Omron Sysmac Studio project Bowery_Farm1 (Sysmac Studio 1.47.0.64008, StandardProject)

# Controller Bowery_Farm1: NJ101-9000 version 1.14
Units and slaves: Node1 : NX-ECC203 (E001); Unit 1 : NX-OD5121 (N1); Unit 2 : NX-SID800 (N2); Unit 3 : NX-SOD400 (N3); Node41 : GX-JC06(IN,X2,X3) Main device (E005); Node8 : NX-ECC203 (LiftGR04); Unit 1 : NX-ID5442 (N9_1); Unit 2 : NX-ID5442 (N10_1); Unit 3 : NX-OD4121 (N11_1); Unit 4 : NX-SID800 (N12_1); Unit 5 : NX-SOD400 (N13_1); Node42 : GX-JC03 (E003); Node43 : NX-ECC203 (E004); Unit 1 : NX-EC0222 (N8_1); Node5 : NX-ECC203 (LiftGR03); Unit 1 : NX-ID5442 (N9); Unit 2 : NX-ID5442 (N10); Unit 3 : NX-OD4121 (N11); Unit 4 : NX-SID800 (N12); Unit 5 : NX-SOD400 (N13); Node32 : GX-JC03 (LiftGR03_Switch); Node33 : NX-ECC203 (LiftGR03_Dek); Unit 1 : NX-EC0222 (N33); Node44 : GX-JC06(X4,X5,X6) Sub-device (E006); Power Supply : NJ-Px3001; CPU : NJ101-9000
Task PrimaryTask (priority 4, period or condition 4000): Mobile_Machines, General, Work_Level01, Work_Mezzanine
Task ReadSettings (priority 8, period or condition 20000): ReadSettings
Library Greencube library 1.2020.1116 (contents left out)

TYPE ST_FB_40401_InputsLift : STRUCT
    LS_FallProtect : BOOL;  (* Limit switch fall protection *)
    LS_Lift_Up : BOOL;  (* Limit switch lift up *)
    LS_Lift_Down : BOOL;  (* Limit switch lift down *)
    LC_Car_Free_Back : BOOL;  (* Photocell carrier detection free backside *)
    LC_Car_Present : BOOL;  (* Photocell carrier present *)
    LC_Car_Free_Front : BOOL;  (* Photocell carrier detection free frontside *)
    LC_Con_Free_Back : BOOL;  (* Photocell container detection free backside *)
    LC_Con_Present : BOOL;  (* Photocell container present *)
    LC_Con_Free_Front : BOOL;  (* Photocell container detection free frontside *)
    IS_Act_Back_Out : BOOL;  (* Inductive sensor actuator backside out *)
    IS_Act_Back_In : BOOL;  (* Inductive sensor actuator backside in *)
    IS_Act_Front_Out : BOOL;  (* Inductive sensor actuator frontside out *)
    IS_Act_Front_In : BOOL;  (* Inductive sensor actuator frontside in *)
    IS_Lift_Level : BOOL;  (* Inductive sensor lift at a level *)
    Clixon_M1 : BOOL;  (* Temperature controller M1 *)
    Clixon_M2 : BOOL;  (* Temperature controller M2 *)
    Clixon_M3 : BOOL;  (* Temperature controller M3 *)
    Clixon_M4 : BOOL;  (* Temperature controller M4 *)
    RC_Tray_Stopper_Min_Back_Up : BOOL;  (* Tray stopper min backside *)
    RC_Tray_Stopper_Max_Back_Up : BOOL;  (* Tray stopper max backside *)
    RC_Tray_Stopper_Min_Front_Up : BOOL;  (* Tray stopper min frontside *)
    RC_Tray_Stopper_Max_Front_Up : BOOL;  (* Tray stopper max frontside *)
    IS_Con_In_Pos_Front : BOOL;  (* Inductive sensor tray is in position front *)
    IS_Con_In_Pos_Back : BOOL;  (* Inductive sensor tray is in position back *)
    LC_Lift_Free_Back : ARRAY[0..15] OF BOOL;  (* Photocell lift free backside Level[i] *)
    LC_Lift_Free_Front : ARRAY[0..15] OF BOOL;  (* Photocell lift free frontside Level[i] *)
    IO_OK : BOOL;  (* Ethercat IO is OK *)
END_STRUCT END_TYPE
TYPE ST_FB_40303_Commands : STRUCT
    SprayBoomToLeft : BOOL;  (* Move sprayboom to left; offset 0.0 *)
    SprayBoomToRight : BOOL;  (* Move sprayboom to right; offset 0.1 *)
    SprayBoomStop : BOOL;  (* Move sprayboom stop; offset 0.2 *)
    LiftingFrame_Up : BOOL;  (* Lifting frame up; offset 1.0 *)
    LiftingFrame_Down : BOOL;  (* Lifting frame down; offset 1.1 *)
    LiftingFrameFirstPush_Up : BOOL;  (* Lifting frame first push up; offset 2.0 *)
    LiftingFrameFirstPush_Down : BOOL;  (* Lifting frame first push down; offset 2.1 *)
    ClampsContainerClose : BOOL;  (* Clamps container close; offset 3.0 *)
    ClampsContainerOpen : BOOL;  (* Clamps container open; offset 3.1 *)
    ClampsBottomLeft_Up : BOOL;  (* Clamps bottom left up; offset 4.0 *)
    ClampsBottomLeft_Down : BOOL;  (* Clamps bottom left down; offset 4.1 *)
    ClampsBottomRight_Up : BOOL;  (* Clamps bottom right up; offset 5.0 *)
    ClampsBottomRight_Down : BOOL;  (* Clamps bottom right down; offset 5.1 *)
    DirtBelt_Forward : BOOL;  (* Dirtbelt forward; offset 6.0 *)
    DirtBelt_Backward : BOOL;  (* Dirtbelt backward; offset 6.1 *)
    DirtBelt_Stop : BOOL;  (* Dirtbelt stop; offset 6.2 *)
    Brush_Forward : BOOL;  (* Brush forward; offset 7.0 *)
    Brush_Backward : BOOL;  (* Brush backward; offset 7.1 *)
    Brush_Stop : BOOL;  (* Brush stop; offset 7.2 *)
    Brush_Fixed : BOOL;  (* Brush fixed; offset 8.0 *)
    Brush_Loose : BOOL;  (* Brush loose; offset 8.1 *)
    SemiAutomatic_StartWashCycle : BOOL;  (* SemiAutomatic, start wash cycle; offset 9.0 *)
    SemiAutomatic_StartCleanBrushCycle : BOOL;  (* SemiAutomatic, start clean brush cycle; offset 9.1 *)
END_STRUCT END_TYPE
TYPE ST_FB_40303_Inputs : STRUCT
    EmergencyStop_OK : BOOL;  (* Emergency stop OK *)
    TurningFrame_Up : BOOL;  (* Lifting frame cilinder is out *)
    TurningFrame_Middle : BOOL;  (* Lifting frame cilinder is in *)
    TurningFrame_Down : BOOL;  (* Lifting frame cilinder is out *)
    Container_Present_1 : BOOL;  (* Container present *)
    Container_Present_2 : BOOL;  (* Container present *)
    Clamp_Container_Fixed_1 : BOOL;  (* Container clamp fixed *)
    Clamp_Container_Loose_1 : BOOL;  (* Container clamp loose *)
    Clamp_Container_Fixed_2 : BOOL;  (* Container clamp fixed *)
    Clamp_Container_Loose_2 : BOOL;  (* Container clamp loose *)
    SprayBoom_Left : BOOL;  (* Sprayboom left *)
    SprayBoom_Right : BOOL;  (* Sprayboom right *)
    SprayBoom_WaterLevel_OK : BOOL;  (* Water float is OK *)
    SprayBoom_WaterLevel_StartFill : BOOL;  (* Water unit in error *)
    InverterStatus_TurningFrame : ST_MX2\Status;  (* Inverter status *)
    InverterStatus_Sprayboom : ST_MX2\Status;  (* Inverter status *)
    InverterStatus_DirtBelt : ST_MX2\Status;  (* Inverter status *)
END_STRUCT END_TYPE
TYPE ST_FB_40303_Outputs : STRUCT
    M_CleanWaterPump : BOOL;  (* Run pump is OK *)
    S_FillCleanWater : BOOL;  (* Valve lifting up *)
    S_CleanWaterDirtBelt : BOOL;  (* Valve lifting down *)
    Actuator_ClampCont_Fixed_1 : BOOL;  (* Valve container fixed *)
    Actuator_ClampCont_Loose_1 : BOOL;  (* Valve container loose *)
    Actuator_ClampCont_Fixed_2 : BOOL;  (* Valve container fixed *)
    Actuator_ClampCont_Loose_2 : BOOL;  (* Valve container loose *)
    Brake_TurningFrame : BOOL;  (* Valve container fixed *)
    SignalLamp_Red : BOOL;  (* Valve bottom clamp fixed (towards container) *)
    SignalLamp_Orange : BOOL;  (* Valve bottom clamp loose *)
    SignalLamp_Green : BOOL;  (* Valve bottom clamp fixed (towards container) *)
    InverterCommands_TurningFrame : ST_MX2\Command;  (* Inverter commands *)
    InverterCommands_Sprayboom : ST_MX2\Command;  (* Inverter commands *)
    InverterCommands_DirtBelt : ST_MX2\Command;  (* Inverter commands *)
    InverterSpeed_TurningFrame : UINT;  (* Inverter speed *)
    InverterSpeed_Sprayboom : UINT;  (* Inverter speed *)
    InverterSpeed_DirtBelt : UINT;  (* Inverter speed *)
END_STRUCT END_TYPE
TYPE ST_FB_40303_Settings : STRUCT
    TurningFrame_Inverter_Parameters : ST_MX2\Parameters;  (* ParameterSet for inverter *)
    TurningFrame_NodeNumber : UINT;  (* Node number inverter *)
    Sprayboom_Inverter_Parameters : ST_MX2\Parameters;  (* ParameterSet for inverter *)
    Sprayboom_NodeNumber : UINT;  (* Node number inverter *)
    DirtBelt_Inverter_Parameters : ST_MX2\Parameters;  (* ParameterSet for inverter *)
    DirtBelt_NodeNumber : UINT;  (* Node number inverter *)
    Sprayboom_Amount_Clean : UINT;  (* Amount of movements to clean container *)
    Sprayboom_Speed : UINT;  (* Minimum speed *)
    Sprayboom_MaxRunTime : UINT;  (* Maximum runtime of the sprayboom *)
    Sprayboom_Delay_SensorRight : UINT;  (* Delay time on sensor right *)
    Sprayboom_Delay_SensorLeft : UINT;  (* Delay time on sensor right *)
    Sprayboom_Time_PressureOn : UINT;  (* Timer pressure sprayboom is low enough after switching on *)
    Sprayboom_Time_PressureOff : UINT;  (* Timer pressure sprayboom is low enough after switching off *)
    Sprayboom_Amount_CleanGutterRight : UINT;  (* Amount of movements to clean gutter begin container *)
    Sprayboom_Amount_CleanGutterLeft : UINT;  (* Amount of movements to clean gutter begin container *)
    Sprayboom_Time_CleanGutterRight : UINT;  (* Pulse value end container sprayboom *)
    Sprayboom_Time_CleanGutterLeft : UINT;  (* Pulse value end container sprayboom *)
    Clamps_TimeOut : UINT;  (* Delay time on sensor out *)
    Clamps_Time_Delay_In : UINT;  (* Delay time on sensor out *)
    Clamps_Time_Delay_Out : UINT;  (* Delay time on sensor out *)
    TurningFrame_Speed_MIN : UINT;  (* Speed for dirtbelt *)
    TurningFrame_Speed_MAX : UINT;  (* Speed for dirtbelt *)
    TurningFrame_TimeOut : UINT;  (* Time before warning is given "does not reach end switch" *)
    TurningFrame_Time_Delay_Down : UINT;  (* Delay time on sensor in *)
    TurningFrame_Time_Delay_Up : UINT;  (* Delay time on sensor out *)
    TurningFrame_Time_Delay_Middle : UINT;  (* Delay time on sensor out *)
    TurningFrame_HighSpeed_Down : UINT;  (* Time movement high speed down *)
    TurningFrame_HighSpeed_Up : UINT;  (* Time movement high speed up *)
    Dirtbelt_Speed : UINT;  (* Speed for dirtbelt *)
    Dirtbelt_RunTimeAfterSpray : UINT;  (* Time that dirtbelt needs to run longer after spraying is stopped *)
END_STRUCT END_TYPE
TYPE ST_FB_40303_Cycle_Turning : STRUCT
    Step00 : BOOL;  (* Request for cleaning, lift middle *)
    Step01 : BOOL;  (* Detect container, close clamps *)
    Step02 : BOOL;  (* Lift up, ready to clean *)
    Step03 : BOOL;  (* Cleaning finished, start lifting down *)
    Step04 : BOOL;  (* Lift down. open container clamps *)
    Step05 : BOOL;  (* Open clamps *)
    Step06 : BOOL;  (* Lift from middle to down *)
    Step07 : BOOL;  (* Container clamps open, communication to external system *)
    Step08 : BOOL;  (* OK from external system, reset cycle *)
END_STRUCT END_TYPE
TYPE ST_FB_40303_Cycle_Cleaning : STRUCT
    Step00 : BOOL;  (* Move sprayboom to begin container *)
    Step01 : BOOL;  (* Put on sprayboom *)
    Step02 : BOOL;  (* Move sprayboom to left side for gutter cleaning *)
    Step03 : BOOL;  (* Move sprayboom to right side for gutter cleaning *)
    Step04 : BOOL;  (* Move sprayboom to clean container *)
    Step07 : BOOL;  (* Put off sprayboom *)
    Step08 : BOOL;  (* Set container status clean, reset cycle *)
END_STRUCT END_TYPE
TYPE ST_Area : STRUCT
    Level : UDINT;  (* Level *)
    X_MIN : UDINT;  (* X minimum value *)
    X_MAX : UDINT;  (* X maximum value *)
    Y_Back : UDINT;  (* Y back value *)
    Y_Front : UDINT;  (* Y front value *)
END_STRUCT END_TYPE
TYPE ST_Settings_CP : STRUCT
    Margin_AreaCompare : UDINT;  (* Margin that is used for area comparison *)
    Setting_Margin_X : UDINT;
    Setting_Margin_Y : UDINT;
END_STRUCT END_TYPE
TYPE ST_XTrack : STRUCT
    XTrack_Number : UINT;  (* Number of the X-Track *)
    MinimumPosition : UDINT;  (* Minimum position *)
    MaximumPosition : UDINT;  (* Maximum position *)
END_STRUCT END_TYPE
TYPE ST_Grant : STRUCT
    Enter : BOOL;  (* Grant Enter; offset 0.0 *)
    Leave : BOOL;  (* Grant Leave; offset 0.1 *)
END_STRUCT END_TYPE
TYPE ST_FB_40401_SettingsLift : STRUCT
    MinimumPulseLevel : UDINT;  (* Minimum pulses the lift can go to *)
    MaximumPulseLevel : UDINT;  (* Maximum pulses the lift can go to *)
    MinimumPosition : UDINT;  (* Minimum floor for this lift *)
    MaximumPosition : UDINT;  (* Maximum floor for this lift *)
    PulseLevel : ARRAY[1..16] OF UDINT;  (* Pulse position for each floor *)
    NeedLevelSensor : ARRAY[1..16] OF BOOL;  (* Need position level sensor *)
    MinimumSpeed : UINT;  (* Minimum elevation speed *)
    MaximumSpeed : UINT;  (* Maximum elevation speed *)
    Dec_Area_High : UDINT;
    Dec_Area_Low : UDINT;
    SafeStopTime : UINT;  (* Time needed to stop safely *)
    Tolerance_At_Position : UDINT;  (* Amount of pulses encoder is allowed to deviate from desired position *)
    ParametersLift : ST_MX2\Parameters;  (* Inverter parameters for lift inverter *)
    NodeNummerLift : UINT;  (* ECat node number of lift inverter *)
    ParametersChain : ST_MX2\Parameters;  (* Inverter parameters for chain inverter *)
    NodeNummerChain : UINT;  (* ECat node number of chain inverter *)
    BrakeReleaseFreq : UINT;  (* Minimum frequency the inverter needs to be for the break to release *)
    ActuatorsLastPosition : BOOL;
    ActuatorBackOn : BOOL;
    ActuatorFrontOn : BOOL;
    PositionReferenceOk : BOOL;
    LoadGateOk : BOOL;
    UnloadGateOk : BOOL;
    MachineCode : UINT;
    ChainHighSpeed : UINT;
    MinimumSpeedChain : UINT;
    MaximumSpeedChain : UINT;
    UseBenchUnloadInstruction : BOOL;
    TimeConFreeBackDON : UINT;
    TimeConFreeBackDOFF : UINT;
    TimeConFreeFrontDON : UINT;
    TimeConFreeFrontDOFF : UINT;
    UnloadToLOcation : UINT;
    Option_InductiveTraydetection : BOOL;
    TimeConInductiveBackDON : UINT;
    TimeConInductiveBackDOFF : UINT;
    TimeConInductiveFrontDON : UINT;
    TimeConInductiveFrontDOFF : UINT;
    Warning_Tolerance_At_Position : UDINT;  (* Amount of pulses encoder is allowed to deviate from desired position for warning *)
    TooFarAllowed : UINT;
    ResetValueMargin : UDINT;
END_STRUCT END_TYPE
TYPE ST_FB_40401_UserSetting : STRUCT
    Overrule_LC_Back : Array[0..15] OF BOOL;
    Overrule_LC_Front : Array[0..15] OF BOOL;
END_STRUCT END_TYPE
TYPE ST_FB_40401_OutputsLift : STRUCT
    Brake_Back : BOOL;  (* Release brake lift *)
    Actuator_Back_Out : BOOL;  (* Lift actuator backside out *)
    Actuator_Back_In : BOOL;  (* Lift actuator backside in *)
    Actuator_Front_Out : BOOL;  (* Lift actuator frontside out *)
    Actuator_Front_In : BOOL;  (* Lift actuator frontside in *)
    Brake_Front : BOOL;  (* Release brake lift *)
    V_TrayStopper_Front_Up : BOOL;  (* Valve traystopper front up *)
    V_Traystopper_Back_Up : BOOL;  (* Valve traystopper back up *)
    LC_Carrier_Free : BOOL;  (* Photocell's carrier detection free *)
    LC_Container_Free : BOOL;  (* Photocell's container detection free *)
END_STRUCT END_TYPE
TYPE ST_FB_40401_Commands : STRUCT
    Move : ST_ManualControl_Actuator;  (* offset 0.0 *)
    Chain : ST_ManualControl_Actuator;  (* offset 2.0 *)
    ActuatorFront : ST_ManualControl_Actuator;  (* offset 4.0 *)
    ActuatorBack : ST_ManualControl_Actuator;  (* offset 6.0 *)
    TraystopperFront : ST_ManualControl_Actuator;  (* offset 8.0 *)
    TraystopperBack : ST_ManualControl_Actuator;  (* offset 10.0 *)
    Semi_DesiredLevel : UINT;  (* Position reference in semi-automatic mode; offset 20.0 *)
    Semi_StartToDesiredLevel : BOOL;  (* Semi_DesiredLevel; offset 22.0 *)
    Calibrate_Level : UINT;  (* Calibrate level; offset 24.0 *)
    Calibrate_SetLevel : BOOL;  (* Calibrate set level; offset 26.0 *)
    MoveFastOn : BOOL;  (* Move fast on; offset 28.0 *)
    MoveFastOff : BOOL;  (* Move fast off; offset 28.1 *)
    MoveFastStatus : BOOL;  (* Move fast status; offset 28.2 *)
    Status_Move : ST_Status_Actuator;  (* offset 30.0 *)
    Status_Chain : ST_Status_Actuator;  (* offset 32.0 *)
    Status_ActuatorFront : ST_Status_Actuator;  (* offset 34.0 *)
    Status_ActuatorBack : ST_Status_Actuator;  (* offset 36.0 *)
    Status_TraystopperFront : ST_Status_Actuator;  (* offset 38.0 *)
    Status_TraystopperBack : ST_Status_Actuator;  (* offset 40.0 *)
END_STRUCT END_TYPE
TYPE ST_FB_40401_Cyc_Move : STRUCT
    Step00 : BOOL;  (* Move instruction, start move actuators to correct position *)
    Step01 : BOOL;  (* Actuators in correct position, start move to reference position *)
    Step02 : BOOL;  (* Lift at position, update actual level carrier *)
    Step03 : BOOL;  (* Carrier level is updated, report job done *)
    Step04 : BOOL;  (* Job done confirmed, reset cycle *)
END_STRUCT END_TYPE
TYPE ST_FB_40401_Cyc_LoadBench : STRUCT
    Step00 : BOOL;  (* Instruction is load bench, check lift level *)
    Step01 : BOOL;  (* Lift is at the right level, start chain conveyer *)
    Step02 : BOOL;  (* Bench is on his way *)
    Step03 : BOOL;  (* Bench is in the right position, do data transfer *)
    Step04 : BOOL;  (* Data transfer is okay, check instruction ready *)
    Step05 : BOOL;  (* Instruction ready, reset cycle *)
    Back : BOOL;  (* Load bench from backside *)
    Front : BOOL;  (* Load bench from frontside *)
END_STRUCT END_TYPE
TYPE ST_FB_40401_Cyc_UnloadBench : STRUCT
    Step00 : BOOL;  (* Instruction is unload bench, check lift level *)
    Step01 : BOOL;  (* Lift is at the right level, start chain conveyer *)
    Step02 : BOOL;  (* Bench is on his way *)
    Step03 : BOOL;  (* Lift is empty, do data transfer *)
    Step04 : BOOL;  (* Data transfer is okay, check instruction ready *)
    Step05 : BOOL;  (* Instruction ready, reset cycle *)
    Back : BOOL;  (* Unload bench from backside *)
    Front : BOOL;  (* Unload bench from frontside *)
END_STRUCT END_TYPE
TYPE ST_FB_40401_Cyc_LoadCarrier : STRUCT
    Step00 : BOOL;  (* Load carrier desired, move actuator down *)
    Step01 : BOOL;  (* Actuator is in position, carrier can move *)
    Step02 : BOOL;  (* Carrier is in position, put actuator up *)
    Step03 : BOOL;  (* Actuator is up, loading carrier is ready *)
    Back : BOOL;  (* Load carrier from backside *)
    Front : BOOL;  (* Load carrier from frontside *)
END_STRUCT END_TYPE
TYPE ST_FB_40401_Cyc_UnloadCarrier : STRUCT
    Step00 : BOOL;  (* Unload carrier desired, move actuator down *)
    Step01 : BOOL;  (* Actuator is in position, carrier can move *)
    Step02 : BOOL;  (* Carrier is out the lift, put actuator up *)
    Step03 : BOOL;  (* Actuator is up, unloading carrier is ready *)
    Back : BOOL;  (* Unload carrier from backside *)
    Front : BOOL;  (* Unload carrier from frontside *)
END_STRUCT END_TYPE
TYPE ST_FB_40401_Cyc_Attach : STRUCT
    Step00 : BOOL;  (* Attach is desired, move actuator out (Stopper down) *)
    Step01 : BOOL;  (* Stopper is down, report job done *)
    Step02 : BOOL;  (* Job done confirmend, reset cycle *)
    Back : BOOL;  (* Attach on the back side *)
    Front : BOOL;  (* Attach on the front side *)
END_STRUCT END_TYPE
TYPE ST_FB_40401_Cyc_Detach : STRUCT
    Step00 : BOOL;  (* Attach is desired, move actuators in (Stoppers up) *)
    Step01 : BOOL;  (* Stoppers are up, report job done *)
    Step02 : BOOL;  (* Job done confirmend, reset cycle *)
END_STRUCT END_TYPE
TYPE ST_FB_40401_CommOut : STRUCT
    SupplySignal : BOOL;  (* offset 0.0 *)
    RequestSignal : BOOL;  (* offset 0.1 *)
    StopOutbound : BOOL;  (* offset 0.3 *)
END_STRUCT END_TYPE
TYPE ST_FB_40401_CommIn : STRUCT
    SupplySignal : BOOL;  (* offset 0.0 *)
    OutboundBusy : BOOL;  (* offset 0.1 *)
    OutboundReady : BOOL;  (* offset 0.2 *)
    RequestSignal : BOOL;  (* offset 0.3 *)
    InboundBusy : BOOL;  (* offset 0.4 *)
    InboundReady : BOOL;  (* offset 0.5 *)
END_STRUCT END_TYPE
TYPE ST_FB_40401_Status : STRUCT
    Lift_With_Bench : BOOL;  (* offset 0.0 *)
    Lift_With_Loaded_Carrier : BOOL;  (* offset 0.1 *)
    Lift_With_Unloaded_Carrier : BOOL;  (* offset 0.2 *)
END_STRUCT END_TYPE
TYPE ST_Manual_Track : STRUCT
    Forward : BOOL;  (* offset 0.0 *)
    Reverse : BOOL;  (* offset 0.1 *)
    Stop : BOOL;  (* offset 0.2 *)
    BridgeUp : BOOL;  (* offset 0.3 *)
    BridgeDown : BOOL;  (* offset 0.4 *)
END_STRUCT END_TYPE
TYPE ST_CP : STRUCT
    Alarm : BOOL;  (* offset 2.0 *)
    Manual : BOOL;  (* offset 2.1 *)
    Busy : BOOL;  (* offset 2.2 *)
    Enable : BOOL;  (* offset 2.3 *)
    Emergencystop : BOOL;  (* offset 2.4 *)
    MachineCycle : UINT;  (* offset 4.0 *)
    Location : UINT;  (* offset 6.0 *)
    MachineNumber : UINT;  (* offset 8.0 *)
    SoftwareVersion : UINT;  (* offset 10.0 *)
    Alarm00 : WORD;  (* offset 12.0 *)
    Alarm01 : WORD;  (* offset 14.0 *)
    Warning00 : WORD;  (* offset 16.0 *)
    ResetAlarm : BOOL;  (* offset 18.1 *)
    ResetCycle : BOOL;  (* offset 18.2 *)
    MachineOn : BOOL;  (* offset 18.4 *)
END_STRUCT END_TYPE
TYPE ST_FB_30050_Inputs : STRUCT
    IS_Track201 : BOOL;
    IS_Track202 : BOOL;
    LS_TrackUp : BOOL;
    LS_TrackDown : BOOL;
    IS_Present : BOOL;
    IS_PB_Run : BOOL;
END_STRUCT END_TYPE
TYPE ST_FB_30050_Settings : STRUCT
    Inverter_Parameters : ST_MX2\Parameters;
    Inverter_NodeNumber : UINT;
    TrackDirection : UINT;
    ForwardIsInput : BOOL;  (* Forward is input over track *)
    MaxSpeed : INT;
    MinSpeed : INT;
    UsePushButton : BOOL;
    TimeDelayON_IS201 : UINT;
    TimeDelayOFF_IS201 : UINT;
    TimeDelayON_IS202 : UINT;
    TimeDelayOFF_IS202 : UINT;
    TimeDelayON_LSTrackUp : UINT;
    TimeDelayON_LSTrackDown : UINT;
    TimeDelayON_ISPresent : UINT;
    TimeDelayOFF_ISPresent : UINT;
    MAX_Run_Time : UINT;
    NoMotor : BOOL;
END_STRUCT END_TYPE
TYPE ST_FB_30050_CommOutPipe : STRUCT
    SupplySignal : BOOL;
    RequestSignal : BOOL;
    SectionIsLow : BOOL;
    StopOutbound : BOOL;
END_STRUCT END_TYPE
TYPE ST_FB_30050_CommInPipe : STRUCT
    SupplySignal : BOOL;
    OutboundBusy : BOOL;
    OutboundReady : BOOL;
    RequestSectionDown : BOOL;
    InboundBusy : BOOL;
    InboundReady : BOOL;
END_STRUCT END_TYPE
TYPE ST_FB_30050_Cyc_Inbound : STRUCT
    Step00 : BOOL;  (* Instruction inbound and bridge is empty, track down *)
    Step01 : BOOL;  (* Track is down, request inbound *)
    Step02 : BOOL;  (* Bench is total at track, do transfer *)
    Step03 : BOOL;  (* Transfer is okay, put track up *)
    Step04 : BOOL;  (* Track is up, reset cycle *)
END_STRUCT END_TYPE
TYPE ST_FB_30050_Cyc_Outbound : STRUCT
    Step00 : BOOL;  (* Request for outbound, track down *)
    Step01 : BOOL;  (* Track is down, do transfer *)
    Step02 : BOOL;  (* Transfer is okay *)
    Step03 : BOOL;  (* request for outbound is gone, reset cycle *)
END_STRUCT END_TYPE
TYPE ST_LIft_TrayCarrier_Info : STRUCT
    CarrierNot_Loaded_Lift1 : BOOL;
    CarrierNot_Loaded_Lift2 : BOOL;
    CarrierNot_Loaded_Lift3 : BOOL;
    CarrierNot_Loaded_Lift4 : BOOL;
    CarrierNot_Loaded_Lift5 : BOOL;
    CarrierNot_Loaded_Lift6 : BOOL;
    CarrierNot_Loaded_Lift7 : BOOL;
    CarrierNot_Loaded_Lift8 : BOOL;
    TrayNot_Loaded_Lift1 : BOOL;
    TrayNot_Loaded_Lift2 : BOOL;
    TrayNot_Loaded_Lift3 : BOOL;
    TrayNot_Loaded_Lift4 : BOOL;
    TrayNot_Loaded_Lift5 : BOOL;
    TrayNot_Loaded_Lift6 : BOOL;
    TrayNot_Loaded_Lift7 : BOOL;
    TrayNot_Loaded_Lift8 : BOOL;
END_STRUCT END_TYPE
TYPE ST_FB_30051_Inputs : STRUCT
    IS_Track201 : BOOL;
    IS_Track202 : BOOL;
    LS_BeltUp : BOOL;
    LS_BeltDown : BOOL;
    IS_Present : BOOL;
    IS_PB_Run : BOOL;
END_STRUCT END_TYPE
TYPE ST_FB_30051_Settings : STRUCT
    Inverter_Parameters_Track : ST_MX2\Parameters;
    Inverter_Parameters_Belt : ST_MX2\Parameters;
    Inverter_NodeNumber_Track : UINT;
    Inverter_NodeNumber_Belt : UINT;
    TrackDirection : UINT;  (* (1 = From buffer, 2 = To buffer) *)
    ForwardIsInput : BOOL;  (* Forward is input over track *)
    MaxSpeed : INT;
    MinSpeed : INT;
    TimeHighSpeed : UINT;
    UsePushButton : BOOL;
    TimeDelayON_IS201 : UINT;
    TimeDelayOFF_IS201 : UINT;
    TimeDelayON_IS202 : UINT;
    TimeDelayOFF_IS202 : UINT;
    TimeDelayON_LSTrackUp : UINT;
    TimeDelayON_LSTrackDown : UINT;
    TimeDelayON_ISPresent : UINT;
    TimeDelayOFF_ISPresent : UINT;
    MAX_Run_Time : UINT;
    UseInstructionTrack : BOOL;
    MinSpeedBelt : INT;
    MaxSpeedBelt : INT;
    TimeHighSpeedBelt : UINT;
    HardwareCodeBuffer : UINT;  (* side of machine where buffer is (eg. 201 or 202) *)
    DoTransferInbound_101 : BOOL;  (* Do transfer inbound from 101 *)
    DoTransferOutbound_101 : BOOL;  (* Do transfer outbound from 101 *)
    DoTransferInbound201_Buffer : BOOL;  (* Do transfer inbound from buffer *)
    DoTransferOutbound201_Buffer : BOOL;  (* Do transfer outbound to buffer *)
    DoTransferInbound202_Buffer : BOOL;  (* Do transfer inbound from buffer *)
    DoTransferOutbound202_Buffer : BOOL;  (* Do transfer outbound to buffer *)
    DoubleSolenoidValve : BOOL;  (* True = Double, False = Single *)
END_STRUCT END_TYPE
TYPE ST_FB_30052_Settings : STRUCT
    Inverter_Parameters_Track : ST_MX2\Parameters;
    Inverter_NodeNumber_Track : UINT;
    TrackDirection : UINT;  (* (1 = From buffer, 2 = To buffer) *)
    ForwardIsInput : BOOL;  (* Forward is input over track *)
    MaxSpeed : INT;
    MinSpeed : INT;
    TimeHighSpeed : UINT;
    TimeDelayON_IS201 : UINT;
    TimeDelayOFF_IS201 : UINT;
    TimeDelayON_IS202 : UINT;
    TimeDelayOFF_IS202 : UINT;
    TimeDelayON_LSTrackUp : UINT;
    TimeDelayON_LSTrackDown : UINT;
    TimeDelayON_ISPresent : UINT;
    TimeDelayOFF_ISPresent : UINT;
    MAX_Run_Time : UINT;
    MinSpeedBelt : INT;
    MaxSpeedBelt : INT;
    TimeHighSpeedBelt : UINT;
    HardwareCodeBuffer : UINT;  (* side of machine where buffer is (eg. 201 or 202) *)
    DoTransferInbound_101 : BOOL;  (* Do transfer inbound from 101 *)
    DoTransferOutbound_101 : BOOL;  (* Do transfer outbound to 101 *)
    DoTransferInbound_Buffer : BOOL;  (* Do transfer inbound from buffer *)
    DoTransferOutbound_Buffer : BOOL;  (* Do transfer outbound to buffer *)
    DoubleSolenoidValve : BOOL;  (* True = Double, False = Single *)
END_STRUCT END_TYPE
TYPE ST_FB_30051_Cyc_Track201 : STRUCT
    Step00 : BOOL;  (* Instruction is from 201. *)
    Step01 : BOOL;  (* Supply signal, do transfer. *)
    Step02 : BOOL;  (* Transfer OK, wait till tray is complete at track. *)
    Step03 : BOOL;  (* Tray is complete at track, wait for tray request from external machine. *)
END_STRUCT END_TYPE
TYPE ST_FB_30051_Cyc_Track202 : STRUCT
    Step00 : BOOL;  (* Instruction is from 202. *)
    Step01 : BOOL;  (* Supply signal, do transfer. *)
    Step02 : BOOL;  (* Transfer OK, Wait till tray is complete at track. *)
    Step03 : BOOL;  (* Tray is complete at track, wait for tray request from external machine. *)
END_STRUCT END_TYPE
TYPE ST_FB_30052_Cyc_Track_Inbound : STRUCT
    Step00 : BOOL;  (* Instruction is from workarea, Lift track up *)
    Step01 : BOOL;  (* Track is up, wait for signal *)
    Step02 : BOOL;  (* Supply signal, do transfer *)
    Step03 : BOOL;  (* Transfer OK, Wait till bench is complete at track *)
    Step04 : BOOL;  (* Bench is complete at track, reset cycle *)
END_STRUCT END_TYPE
TYPE ST_FB_30052_Cyc_Track_Outbound : STRUCT
    Step00 : BOOL;  (* Instruction is to workarea, Lift track up *)
    Step01 : BOOL;  (* Track is up, wait for signal *)
    Step02 : BOOL;  (* Supply signal, do transfer *)
    Step03 : BOOL;  (* Transfer OK, Wait till bench is complete at track *)
    Step04 : BOOL;  (* Bench is complete off track, reset cycle *)
END_STRUCT END_TYPE
TYPE ST_FB_30051_CommOutPipe : STRUCT
    SupplySignal : BOOL;
    RequestSignal : BOOL;
    SectionIsLow : BOOL;
    StopOutbound : BOOL;
END_STRUCT END_TYPE
TYPE ST_FB_30051_CommOut201 : STRUCT
    SupplySignal : BOOL;
    RequestSignal : BOOL;
END_STRUCT END_TYPE
TYPE ST_FB_30051_CommOut202 : STRUCT
    SupplySignal : BOOL;
    RequestSignal : BOOL;
END_STRUCT END_TYPE
TYPE ST_FB_30051_CommInPipe : STRUCT
    SupplySignal : BOOL;  (* Supply available for supply from pipeline. *)
    OutboundBusy : BOOL;  (* Machine outbound from pipeline is in progress. *)
    OutboundReady : BOOL;  (* Machine outbound from pipeline is ready. *)
    RequestBridgeUp : BOOL;  (* Request bridge up / section down. *)
    InboundBusy : BOOL;  (* Machine inbound to pipeline is in progress. *)
    InboundReady : BOOL;  (* Machine inbound to pipeline is ready. *)
END_STRUCT END_TYPE
TYPE ST_FB_30051_CommIn201 : STRUCT
    SupplySignal : BOOL;
    RequestSignal : BOOL;
END_STRUCT END_TYPE
TYPE ST_FB_30051_CommIn202 : STRUCT
    SupplySignal : BOOL;
    RequestSignal : BOOL;
END_STRUCT END_TYPE
TYPE ST_FB_30051_Cyc_Inbound : STRUCT
    Step00 : BOOL;  (* Instruction inbound and Track is empty, Belt up *)
    Step01 : BOOL;  (* Belt is up, request inbound *)
    Step02 : BOOL;  (* Bench is total at track, do transfer *)
    Step03 : BOOL;  (* Transfer is okay, put belt down *)
    Step04 : BOOL;  (* Belt is down, reset cycle *)
END_STRUCT END_TYPE
TYPE ST_FB_30051_Cyc_Outbound : STRUCT
    Step00 : BOOL;  (* Request for outbound, belt up *)
    Step01 : BOOL;  (* Belt is up, do transfer *)
    Step02 : BOOL;  (* Transfer is okay *)
    Step03 : BOOL;  (* request for outbound is gone, reset cycle *)
END_STRUCT END_TYPE
TYPE ST_FB_30051_Outputs : STRUCT
    V_Belt_Up : BOOL;
    V_Belt_Down : BOOL;  (* Only with setting DoubleSolenoidValve is TRUE *)
END_STRUCT END_TYPE
TYPE ST_FB_30052_Outputs : STRUCT
    V_Track_Up : BOOL;
    V_Track_Down : BOOL;  (* Only with setting DoubleSolenoidValve is TRUE *)
END_STRUCT END_TYPE
TYPE ST_FB_30051_Commands : STRUCT
    Track_Forward : BOOL;  (* offset 0.0 *)
    Track_Reverse : BOOL;  (* offset 0.1 *)
    Track_Stop : BOOL;  (* offset 0.2 *)
    BeltUp : BOOL;  (* offset 0.3 *)
    BeltDown : BOOL;  (* offset 0.4 *)
    Belt_Forward : BOOL;  (* offset 0.5 *)
    Belt_Reverse : BOOL;  (* offset 0.6 *)
    Belt_Stop : BOOL;  (* offset 0.7 *)
END_STRUCT END_TYPE
TYPE ST_Stacker_Commands : STRUCT
    Track_Forward : BOOL;  (* offset 0.0 *)
    Track_Reverse : BOOL;  (* offset 0.1 *)
    Track_Stop : BOOL;  (* offset 0.2 *)
    StackerUp : BOOL;  (* offset 0.3 *)
    StackerDown : BOOL;  (* offset 0.4 *)
    StackerStop : BOOL;  (* offset 0.5 *)
END_STRUCT END_TYPE
TYPE ST_Stacker_Cyc_Load : STRUCT
    Step00 : BOOL;
    Step01 : BOOL;
    Step02 : BOOL;
    Step03 : BOOL;
    Step04 : BOOL;
    Step05 : BOOL;
    Step06 : BOOL;
    Step07 : BOOL;
    Step08 : BOOL;
END_STRUCT END_TYPE
TYPE ST_Stacker_Cyc_Unload : STRUCT
    Step00 : BOOL;
    Step01 : BOOL;
    Step02 : BOOL;
    Step03 : BOOL;
    Step04 : BOOL;
    Step05 : BOOL;
    Step06 : BOOL;
    Step07 : BOOL;
    Step08 : BOOL;
END_STRUCT END_TYPE
TYPE ST_W03_Cyc : STRUCT
    Step00 : BOOL;  (* Instruction accepted, lower belts W03 and W05 *)
    Step01 : BOOL;  (* Belts down, wait for supply lift *)
    Step02 : BOOL;  (* Supply lift, start belt *)
    Step03 : BOOL;  (* Container completely on belt, lift W03 and W05 if Cleaner is free else reset cycle *)
    Step04 : BOOL;  (* System up, reset cycle *)
END_STRUCT END_TYPE
TYPE ST_W04_Cyc : STRUCT
    Step00 : BOOL;  (* Instruction accepted, lower belt *)
    Step01 : BOOL;  (* Belt is down, wait for supply *)
    Step02 : BOOL;  (* Supply W03, Do transfer *)
    Step03 : BOOL;  (* Transfer OK, start belt *)
    Step04 : BOOL;  (* Container completely on belt, start cleaner *)
    Step04_sub00 : BOOL;  (* Cleaner started, transfer to cleaner *)
    Step04_sub01 : BOOL;  (* Transfer OK, wait for cleaner to be almost ready *)
    Step04_sub02 : BOOL;  (* Cleaner (almost) ready, transfer back to W04 *)
    Step04_sub03 : BOOL;  (* Transfer OK, wait for cleaner to be ready *)
    Step05 : BOOL;  (* Cleaner is ready, lift belt *)
    Step06 : BOOL;  (* Belt up, give supply signal to W05 *)
    Step07 : BOOL;  (* Belt is empty, reset cycle *)
END_STRUCT END_TYPE
TYPE ST_W05_Cyc : STRUCT
    Step00 : BOOL;  (* Instruction accepted, lower belt *)
    Step01 : BOOL;  (* Belt is down, wait for suppy *)
    Step02 : BOOL;  (* Supply from W04, Do transfer *)
    Step03 : BOOL;  (* Transfer OK, start belt *)
    Step04 : BOOL;  (* Container completely on belt, release W04 *)
    Step05 : BOOL;  (* Belt empty, reset cycle *)
END_STRUCT END_TYPE

VAR_GLOBAL
    Status_Lift03 : ST_MX2\Status;  (* at ECAT://node#6/Status *)
    Commands_Lift03 : ST_MX2\Command;  (* at ECAT://node#6/Command *)
    Speed_Lift03 : UINT;  (* at ECAT://node#6/Frequency reference *)
    Inputs_Lift03 : ST_MX2\Input;  (* at ECAT://node#6/d005 Multi-function Input Monitor *)
    Freq_Lift03 : UINT;  (* at ECAT://node#6/Output frequency monitor *)
    N33_Ch1_Encoder_Preset_Position : DINT;  (* at ECAT://node#[33,1]/Ch1 Encoder Present Position *)
    N33_Ch1_Preset_Execution : BOOL;  (* at ECAT://node#[33,1]/Ch1 Encoder Counter Operation Command/Ch1 Preset Execution *)
    N33_Ch1_Preset_Command_Value : DINT;  (* at ECAT://node#[33,1]/Ch1 Preset Command Value *)
    Drive_Rack_Desired_Backward : BOOL;
    Drive_Rack_Desired_Forward : BOOL;
    Drive_Rack_Desired_Reference : BOOL;
    Drive_Rack_ExtraStrong : BOOL;
    Drive_Rack_MaxSpeed : UINT;
    Drive_Rack_Reference : UDINT;
    N005O400 : BOOL;  (* Brake1_Lift03; at ECAT://node#[5,3]/Output Bit 8 bits/Output Bit 00 *)
    N005O405 : BOOL;  (* Brake2_Lift03; at ECAT://node#[5,3]/Output Bit 8 bits/Output Bit 05 *)
    Commands_Lift04 : ST_MX2\Command;  (* at ECAT://node#9/Command *)
    Speed_Lift04 : UINT;  (* at ECAT://node#9/Frequency reference *)
    Status_Lift04 : ST_MX2\Status;  (* at ECAT://node#9/Status *)
END_VAR
VAR_GLOBAL RETAIN
    Supply_Stacker AT %D00006.00 : BOOL;  (* Sensor Dat-A-Control: Supply from stacker *)
    Insert_Stacker AT %D00006.01 : BOOL;  (* Sensor Dat-A-Control: Supply into stacker *)
    T01W01_Loaded AT %D00006.02 : BOOL;
    T01W02_Loaded AT %D00006.03 : BOOL;
    T02W06_Loaded AT %D00006.04 : BOOL;
    LC_Lift3_Disable_Back_Level0 AT %D00007.00 : BOOL;
    LC_Lift3_Disable_Back_Level4 AT %D00007.01 : BOOL;
    LC_Lift3_Disable_Front_Level0 AT %D00007.02 : BOOL;
    LC_Lift3_Disable_Front_Level1 AT %D00007.03 : BOOL;
    LC_Lift3_Disable_Front_Level2 AT %D00007.04 : BOOL;
    LC_Lift3_Disable_Front_Level3 AT %D00007.05 : BOOL;
    LC_Lift3_Disable_Front_Level4 AT %D00007.06 : BOOL;
    LC_Lift3_Disable_Front_Level5 AT %D00007.07 : BOOL;
    Comm_To_Carrier04_SENDREC AT %D06400 : ARRAY[0..199] OF WORD;  (* Comm from Carrier04 (For send/recieve) *)
    Comm_To_Carrier04 AT %D06400 : ST_FB_40701\Comm_IN;  (* ST Comm from Carrier04 *)
    Comm_From_Carrier04_SENDREC AT %D06600 : ARRAY[0..199] OF WORD;  (* Comm from Carrier04 (For send/recieve) *)
    Comm_From_Carrier03_SENDREC AT %D06200 : ARRAY[0..199] OF WORD;  (* Comm from Carrier03 (For send/recieve) *)
    W03_Dat_A_Control AT %D20200 : ST_DatAControl_Standard;  (* Dat a control interface *)
    W03_Commands AT %D20217 : ST_FB_25050\Commands;  (* Commands W03 *)
    W04_Dat_A_Control AT %D20240 : ST_DatAControl_Standard;  (* Dat a control interface *)
    W04_Commands AT %D20257 : ST_FB_25050\Commands;  (* Commands W04 *)
    W05_Dat_A_Control AT %D20280 : ST_DatAControl_Standard;  (* Dat a control interface *)
    W05_Commands AT %D20297 : ST_FB_25050\Commands;  (* Commands W05 *)
    Cleaner_Dat_A_Control AT %D20520 : ST_DatAControl_Standard;  (* Dat a control interface *)
END_VAR
VAR_GLOBAL
    Freq_Lift04 : UINT;  (* at ECAT://node#9/Output frequency monitor *)
    Inputs_Lift04 : ST_MX2\Input;  (* at ECAT://node#9/d005 Multi-function Input Monitor *)
    N005I0308 : BOOL;  (* Knop_Ok_Lift3; at ECAT://node#[5,2]/Input Bit 16 bits/Input Bit 08 *)
    N005I0309 : BOOL;  (* Knop_FW_Lift03(Up); at ECAT://node#[5,2]/Input Bit 16 bits/Input Bit 09 *)
    N005I0310 : BOOL;  (* Knop_Snel_Lift03; at ECAT://node#[5,2]/Input Bit 16 bits/Input Bit 10 *)
    N005I0311 : BOOL;  (* Knop_RV_Lift03(Down); at ECAT://node#[5,2]/Input Bit 16 bits/Input Bit 11 *)
    N005O407 : BOOL;  (* Led_Knop_Ok_Lift1; at ECAT://node#[5,3]/Output Bit 8 bits/Output Bit 07 *)
    N33_Ch1_Counter_Enable : BOOL;  (* at ECAT://node#[33,1]/Ch1 Encoder Counter Operation Command/Ch1 Counter Enable *)
    N005O406 : BOOL;  (* Led_RS_Extern; at ECAT://node#[5,3]/Output Bit 8 bits/Output Bit 06 *)
    SafetyRelays_Lift03 : BOOL;  (* at ECAT://node#[5,5]/Standard Input 1st Byte/So00 Monitor Value *)
    SafetyRelays_Lift04 : BOOL;  (* at ECAT://node#[8,5]/Standard Input 1st Byte/So00 Monitor Value *)
    Commands_Lift03_Ch : ST_MX2\Command;  (* at ECAT://node#7/Command *)
    Speed_Lift03_Ch : UINT;  (* at ECAT://node#7/Frequency reference *)
    Status_Lift03_Ch : ST_MX2\Status;  (* at ECAT://node#7/Status *)
    Freq_Lift03_Ch : UINT;  (* at ECAT://node#7/Output frequency monitor *)
    Inputs_Lift03_Ch : ST_MX2\Input;  (* at ECAT://node#7/d005 Multi-function Input Monitor *)
    Commands_Lift04_Ch : ST_MX2\Command;  (* at ECAT://node#10/Command *)
    Speed_Lift04_Ch : UINT;  (* at ECAT://node#10/Frequency reference *)
    Status_Lift04_Ch : ST_MX2\Status;  (* at ECAT://node#10/Status *)
    Freq_Lift04_Ch : UINT;  (* at ECAT://node#10/Output frequency monitor *)
    Inputs_Lift04_Ch : ST_MX2\Input;  (* at ECAT://node#10/d005 Multi-function Input Monitor *)
    N005O401 : BOOL;  (* Actuator_Back_Out_Lift03; at ECAT://node#[5,3]/Output Bit 8 bits/Output Bit 01 *)
    N005O402 : BOOL;  (* Actuator_Back_In_Lift03; at ECAT://node#[5,3]/Output Bit 8 bits/Output Bit 02 *)
    N005O403 : BOOL;  (* Actuator_Front_Out_Lift03; at ECAT://node#[5,3]/Output Bit 8 bits/Output Bit 03 *)
    N005O404 : BOOL;  (* Actuator_Front_In_Lift03; at ECAT://node#[5,3]/Output Bit 8 bits/Output Bit 04 *)
    I_EStop_OK : BOOL;  (* Emergency stop is OK *)
    ES_OK : BOOL;  (* Emergency stop OK *)
    Trig_ReadSettings : BOOL;
END_VAR
VAR_GLOBAL RETAIN
    Comm_To_Carrier01 AT %D01000 : ST_FB_40701\Comm_IN;  (* ST Comm to Carrier01 *)
    Comm_To_Carrier01_SENDREC AT %D01000 : ARRAY[0..199] OF WORD;  (* Comm to Carrier01 (For send/recieve) *)
END_VAR
VAR_GLOBAL
    N008I0200 : BOOL;  (* Lift04_LS_FallProtect; at ECAT://node#[8,1]/Input Bit 16 bits/Input Bit 00 *)
    N008I0201 : BOOL;  (* Lift04_LS_Up; at ECAT://node#[8,1]/Input Bit 16 bits/Input Bit 01 *)
    N008I0202 : BOOL;  (* Lift04_LS_Down; at ECAT://node#[8,1]/Input Bit 16 bits/Input Bit 02 *)
    N008I0203 : BOOL;  (* Lift04_LC_Car_Free_Back; at ECAT://node#[8,1]/Input Bit 16 bits/Input Bit 03 *)
    N008I0204 : BOOL;  (* Lift04_LC_Car_Pres; at ECAT://node#[8,1]/Input Bit 16 bits/Input Bit 04 *)
    N008I0205 : BOOL;  (* Lift04_LC_Con_Free_Front; at ECAT://node#[8,1]/Input Bit 16 bits/Input Bit 05 *)
    N008I0206 : BOOL;  (* Lift04_LC_Con_Free_Back; at ECAT://node#[8,1]/Input Bit 16 bits/Input Bit 06 *)
    N008I0207 : BOOL;  (* Lift04_Pallet_Pres; at ECAT://node#[8,1]/Input Bit 16 bits/Input Bit 07 *)
    N008I0208 : BOOL;  (* Lift04_LC_Con_Free_Front; at ECAT://node#[8,1]/Input Bit 16 bits/Input Bit 08 *)
    N008I0209 : BOOL;  (* Lift04_NO_Act_Back_Out; at ECAT://node#[8,1]/Input Bit 16 bits/Input Bit 09 *)
    N008I0210 : BOOL;  (* Lift04_NO_Act_Back_In; at ECAT://node#[8,1]/Input Bit 16 bits/Input Bit 10 *)
    N008I0211 : BOOL;  (* Lift04_NO_Act_Front_Out; at ECAT://node#[8,1]/Input Bit 16 bits/Input Bit 11 *)
    N008I0212 : BOOL;  (* Lift04_NO_Ack_Front_In; at ECAT://node#[8,1]/Input Bit 16 bits/Input Bit 12 *)
    N008I0213 : BOOL;  (* Lift04_LC_Lift_Level; at ECAT://node#[8,1]/Input Bit 16 bits/Input Bit 13 *)
    N008I0214 : BOOL;  (* Spare; at ECAT://node#[8,1]/Input Bit 16 bits/Input Bit 14 *)
    N008I0215 : BOOL;  (* Spare; at ECAT://node#[8,1]/Input Bit 16 bits/Input Bit 15 *)
    N008I0300 : BOOL;  (* Lift04_LC_Free_Back01; at ECAT://node#[8,2]/Input Bit 16 bits/Input Bit 00 *)
    N008I0301 : BOOL;  (* Lift04_LC_Free_Back02; at ECAT://node#[8,2]/Input Bit 16 bits/Input Bit 01 *)
    N008I0302 : BOOL;  (* Lift04_LC_Free_Back03; at ECAT://node#[8,2]/Input Bit 16 bits/Input Bit 02 *)
    N008I0303 : BOOL;  (* Lift04_LC_Free_Back04; at ECAT://node#[8,2]/Input Bit 16 bits/Input Bit 03 *)
    N008I0304 : BOOL;  (* Lift04_LC_Free_Back05; at ECAT://node#[8,2]/Input Bit 16 bits/Input Bit 04 *)
    N008I0305 : BOOL;  (* Lift04_LC_Free_Back06; at ECAT://node#[8,2]/Input Bit 16 bits/Input Bit 05 *)
    N008I0306 : BOOL;  (* Lift04_LC_Free_Back07; at ECAT://node#[8,2]/Input Bit 16 bits/Input Bit 06 *)
    N008I0307 : BOOL;  (* Lift04_LC_Free_Back08; at ECAT://node#[8,2]/Input Bit 16 bits/Input Bit 07 *)
    N008I0308 : BOOL;  (* Knop_Ok_Lift04; at ECAT://node#[8,2]/Input Bit 16 bits/Input Bit 08 *)
    N008I0309 : BOOL;  (* Knop_FW_Lift04(Up); at ECAT://node#[8,2]/Input Bit 16 bits/Input Bit 09 *)
    N008I0310 : BOOL;  (* Knop_Snel_Lift04; at ECAT://node#[8,2]/Input Bit 16 bits/Input Bit 10 *)
    N008I0311 : BOOL;  (* Knop_RV_Lift04(Down); at ECAT://node#[8,2]/Input Bit 16 bits/Input Bit 11 *)
    N008I0312 : BOOL;  (* Lift04_LC_Free_Front_05; at ECAT://node#[8,2]/Input Bit 16 bits/Input Bit 12 *)
    N008I0313 : BOOL;  (* Lift04_LC_Free_Front_06; at ECAT://node#[8,2]/Input Bit 16 bits/Input Bit 13 *)
    N008I0314 : BOOL;  (* Lift04_LC_Free_Front_07; at ECAT://node#[8,2]/Input Bit 16 bits/Input Bit 14 *)
    N008I0315 : BOOL;  (* Lift04_LC_Free_Front_08; at ECAT://node#[8,2]/Input Bit 16 bits/Input Bit 15 *)
    N008O0400 : BOOL;  (* Lift04_Brake1; at ECAT://node#[8,3]/Output Bit 8 bits/Output Bit 00 *)
    N008O0401 : BOOL;  (* Lift04_Actuator_Back_Out; at ECAT://node#[8,3]/Output Bit 8 bits/Output Bit 01 *)
    N008O0402 : BOOL;  (* Lift04_Actuator_Back_In; at ECAT://node#[8,3]/Output Bit 8 bits/Output Bit 02 *)
    N008O0403 : BOOL;  (* Lift04_Actuator_Front_Out; at ECAT://node#[8,3]/Output Bit 8 bits/Output Bit 03 *)
    N008O0404 : BOOL;  (* Lift04_Actuator_Front_In; at ECAT://node#[8,3]/Output Bit 8 bits/Output Bit 04 *)
    N008O0405 : BOOL;  (* Lift04_Break2; at ECAT://node#[8,3]/Output Bit 8 bits/Output Bit 05 *)
    N008O0406 : BOOL;  (* Spare; at ECAT://node#[8,3]/Output Bit 8 bits/Output Bit 06 *)
    Led_RS_Extern : BOOL;  (* LED Reset button Estop *)
END_VAR
VAR_GLOBAL RETAIN
    TransferBuffer AT %D00010 : ST_TransferBuffer;  (* TransferBuffer *)
END_VAR
VAR_GLOBAL
    CommSend_Ca01 : BOOL;  (* Communication send to Carrier01 *)
    CommSend_Ca02 : BOOL;  (* Communication send to Carrier02 *)
    CommReceive_Ca01 : BOOL;  (* Communication receive from Carrier01 *)
    CommReceive_Ca02 : BOOL;  (* Communication receive from Carrier02 *)
END_VAR
VAR_GLOBAL RETAIN
    DatAControl_Lift04 AT %D02200 : ST_DatAControl_Standard;  (* Base adress lift 04 *)
    Pocket_Lift03 AT %D01850 : ST_FB_40401_Commands;
    Pocket_Lift04 AT %D02250 : ST_FB_40401_Commands;
END_VAR
VAR_GLOBAL
    Dummy : BOOL;  (* Dummy *)
    N005I0312 : BOOL;  (* Lift03_LC_Free_Front05; at ECAT://node#[5,2]/Input Bit 16 bits/Input Bit 12 *)
    N005I0313 : BOOL;  (* Lift03_1LC_Free_Front06; at ECAT://node#[5,2]/Input Bit 16 bits/Input Bit 13 *)
    N005I0314 : BOOL;  (* Lift03_LC_Free_Front07; at ECAT://node#[5,2]/Input Bit 16 bits/Input Bit 14 *)
    N005I0315 : BOOL;  (* Lift03_LC_Free_Front08; at ECAT://node#[5,2]/Input Bit 16 bits/Input Bit 15 *)
    N33_NX_Unit_I_O_Data_Active_Status : ARRAY[0..63] OF BOOL;  (* at ECAT://node#33/NX Unit I/O Data Active Status 63 *)
    N8_NX_Unit_I_O_Data_Active_Status : ARRAY[0..63] OF BOOL;  (* at ECAT://node#8/NX Unit I/O Data Active Status 63 *)
    N8_Ch1_Counter_Enable : BOOL;  (* at ECAT://node#[43,1]/Ch1 Encoder Counter Operation Command/Ch1 Counter Enable *)
    N8_Ch1_Preset_Command_Value : DINT;  (* at ECAT://node#[43,1]/Ch1 Preset Command Value *)
    N8_Ch1_Preset_Execution : BOOL;  (* at ECAT://node#[43,1]/Ch1 Encoder Counter Operation Command/Ch1 Preset Execution *)
    N8_Ch1_Encoder_Preset_Position : DINT;  (* at ECAT://node#[43,1]/Ch1 Encoder Present Position *)
END_VAR
VAR_GLOBAL RETAIN
    Comm_From_Carrier01 AT %D01200 : ST_FB_40701\Comm_OUT;  (* ST Comm from Carrier01 *)
    Comm_From_Carrier01_SENDREC AT %D01200 : ARRAY[0..199] OF WORD;  (* Comm from Carrier01 (For send/recieve) *)
    Comm_From_Carrier02_SENDREC AT %D01600 : ARRAY[0..199] OF WORD;  (* Comm from Carrier02 (For send/recieve) *)
    Comm_From_Carrier02 AT %D01600 : ST_FB_40701\Comm_OUT;  (* ST Comm from Carrier02 *)
END_VAR
VAR_GLOBAL
    N005I0200 : BOOL;  (* Lift03_LS_FallProtect; at ECAT://node#[5,1]/Input Bit 16 bits/Input Bit 00 *)
    N005I0201 : BOOL;  (* Lift03_LS_Up; at ECAT://node#[5,1]/Input Bit 16 bits/Input Bit 01 *)
    N005I0202 : BOOL;  (* Lift03_LS_Down; at ECAT://node#[5,1]/Input Bit 16 bits/Input Bit 02 *)
    N005I0203 : BOOL;  (* Lift03_LC_Car_Free_Back; at ECAT://node#[5,1]/Input Bit 16 bits/Input Bit 03 *)
    N005I0204 : BOOL;  (* Lift03_LC_Car_Pres; at ECAT://node#[5,1]/Input Bit 16 bits/Input Bit 04 *)
    N005I0205 : BOOL;  (* Lift03_LC_Con_Free_Front; at ECAT://node#[5,1]/Input Bit 16 bits/Input Bit 05 *)
    N005I0206 : BOOL;  (* Lift03_LC_Con_Free_Back; at ECAT://node#[5,1]/Input Bit 16 bits/Input Bit 06 *)
    N005I0207 : BOOL;  (* Lift03_LC_Pallet_Pres; at ECAT://node#[5,1]/Input Bit 16 bits/Input Bit 07 *)
    N005I0208 : BOOL;  (* Lift03_LC_Con_Free_Front; at ECAT://node#[5,1]/Input Bit 16 bits/Input Bit 08 *)
    N005I0209 : BOOL;  (* Lift03_NO_Act_Back_Out; at ECAT://node#[5,1]/Input Bit 16 bits/Input Bit 09 *)
    N005I0210 : BOOL;  (* Lift03_NO_Act_Back_In; at ECAT://node#[5,1]/Input Bit 16 bits/Input Bit 10 *)
    N005I0211 : BOOL;  (* Lift03_NO_Act_Front_Out; at ECAT://node#[5,1]/Input Bit 16 bits/Input Bit 11 *)
    N005I0212 : BOOL;  (* Lift03_NO_Act_Front_In; at ECAT://node#[5,1]/Input Bit 16 bits/Input Bit 12 *)
    N005I0213 : BOOL;  (* Lift03_LC_Lift_Level; at ECAT://node#[5,1]/Input Bit 16 bits/Input Bit 13 *)
    N005I0214 : BOOL;  (* Spare; at ECAT://node#[5,1]/Input Bit 16 bits/Input Bit 14 *)
    N005I0215 : BOOL;  (* Spare; at ECAT://node#[5,1]/Input Bit 16 bits/Input Bit 15 *)
    N005I0300 : BOOL;  (* Lift03_LC_Free_Back01; at ECAT://node#[5,2]/Input Bit 16 bits/Input Bit 00 *)
    N005I0301 : BOOL;  (* Lift03_LC_Free_Back02; at ECAT://node#[5,2]/Input Bit 16 bits/Input Bit 01 *)
    N005I0302 : BOOL;  (* Lift03_LC_Free_Back03; at ECAT://node#[5,2]/Input Bit 16 bits/Input Bit 02 *)
    N005I0303 : BOOL;  (* Lift03_LC_Free_Back04; at ECAT://node#[5,2]/Input Bit 16 bits/Input Bit 03 *)
    N005I0304 : BOOL;  (* Lift03_LC_Free_Back05; at ECAT://node#[5,2]/Input Bit 16 bits/Input Bit 04 *)
    N005I0305 : BOOL;  (* Lift03_LC_Free_Back06; at ECAT://node#[5,2]/Input Bit 16 bits/Input Bit 05 *)
    N005I0306 : BOOL;  (* Lift03_LC_Free_Back07; at ECAT://node#[5,2]/Input Bit 16 bits/Input Bit 06 *)
    N005I0307 : BOOL;  (* Lift03_LC_Free_Back08; at ECAT://node#[5,2]/Input Bit 16 bits/Input Bit 07 *)
    N008O0407 : BOOL;  (* Led_Knop_Ok_Lift04; at ECAT://node#[8,3]/Output Bit 8 bits/Output Bit 07 *)
END_VAR
VAR_GLOBAL RETAIN
    Comm_To_Carrier02 AT %D01400 : ST_FB_40701\Comm_IN;  (* ST Comm to Carrier02 *)
    Comm_To_Carrier02_SENDREC AT %D01400 : ARRAY[0..199] OF WORD;  (* Comm to Carrier02 (For send/recieve) *)
    XTrack_XYPositions_Array AT %D05000 : ARRAY[0..199] OF UINT;
    Lift_Array AT %D05500 : ARRAY[0..99] OF UINT;
END_VAR
VAR_GLOBAL
    FixedLoadPosition_Array : ARRAY[0..199] OF UINT;
    FixedUnloadPosition_Array : ARRAY[0..199] OF UINT;
END_VAR
VAR_GLOBAL RETAIN
    Settings_CP AT %D02500 : ST_Settings_CP;  (* Settings in CP *)
    Area AT %D10000 : ARRAY[0..99] OF ST_Area;  (* Area data *)
    PositionInformation_Rack AT %D00900 : ST_FB_40701\PositionInformation_Rack;
    PositionInformation_Rough AT %D00900 : ARRAY[0..9] OF UINT;
    XTrack_Y_Values AT %D05100 : ARRAY[0..49] OF UDINT;
    PositionInformation_XTrack AT %D00900 : ST_FB_40701\PositionInformation_XTrack;
    XTrack AT %D11000 : ARRAY[0..49] OF ST_XTrack;  (* X-Tracks *)
    Grants AT %E0_00000 : ARRAY[0..9999] OF ST_Grant;  (* Array of grants *)
    XTrack_X_Values AT %D05000 : ARRAY[0..49] OF UDINT;  (* X-Track X values *)
    GrantEnter_Ca01 AT %D00991.00 : BOOL;  (* Grant Enter carrier01 self *)
    GrantLeave_Ca01 AT %D00991.01 : BOOL;  (* Grant Leave carrier01 self *)
    ReservationDB AT %D00600 : ARRAY[0..20] OF ST_FB_Reservation_Carrier;
    RegistrationData_Carrier01 AT %D07000 : ARRAY[0..199] OF UINT;  (* Registration data *)
    RegistrationData_Carrier02 AT %D07200 : ARRAY[0..199] OF UINT;  (* Registration data *)
    RegistrationData_Carrier03 AT %D07400 : ARRAY[0..199] OF UINT;  (* Registration data *)
END_VAR
VAR_GLOBAL
    DstNetAdr_Ca01 : _sDNET_ADR;  (* Send adress Carrier01 *)
    Option_Ca01 : _sRESPONSE;  (* Send options Carrier01 *)
    DstNetAdr_Ca02 : _sDNET_ADR;  (* Send adress Carrier02 *)
    Option_Ca02 : _sRESPONSE;  (* Send options Carrier02 *)
END_VAR
VAR_GLOBAL RETAIN
    GrantEnter_Ca02 AT %D00992.00 : BOOL;  (* Grant Enter carrier02 self *)
    GrantLeave_Ca02 AT %D00992.01 : BOOL;  (* Grant Leave carrier02 self *)
    Lift AT %D05500 : ARRAY[0..9] OF ST_LiftInformation;  (* Lift information *)
    Transfer_BenchSize AT %D00017 : UINT;
    DatAControl_Lift03 AT %D01800 : ST_DatAControl_Standard;  (* Base adress lift 03 *)
    W02_Dat_A_Control AT %D20000 : ST_DatAControl_Standard;
    W02_Commands AT %D20017 : ST_FB_25050\Commands;
END_VAR
VAR_GLOBAL
    N000O0100 : BOOL;  (* Charger_4D402; at ECAT://node#[1,1]/Output Bit 16 bits/Output Bit 00 *)
    N000O0101 : BOOL;  (* Charger_4D102; at ECAT://node#[1,1]/Output Bit 16 bits/Output Bit 01 *)
    N000O0102 : BOOL;  (* LampGreen; at ECAT://node#[1,1]/Output Bit 16 bits/Output Bit 02 *)
    InverterCommands_T01W01 : ST_MX2\Command;  (* at ECAT://node#16/Command *)
    InverterSpeed_T01W01 : INT;  (* at ECAT://node#16/Frequency reference *)
    InverterOutputs_T01W01 : ST_MX2\Output;  (* at ECAT://node#16/Output terminal setting *)
    InverterStatus_T01W01 : ST_MX2\Status;  (* at ECAT://node#16/Status *)
    InverterInputs_T01W01 : ST_MX2\Input;  (* at ECAT://node#16/d005 Multi-function Input Monitor *)
    InverterCommands_T01W02 : ST_MX2\Command;  (* at ECAT://node#11/Command *)
    InverterSpeed_T01W02 : INT;  (* at ECAT://node#11/Frequency reference *)
    InverterOutputs_T01W02 : ST_MX2\Output;  (* at ECAT://node#11/Output terminal setting *)
    InverterStatus_T01W02 : ST_MX2\Status;  (* at ECAT://node#11/Status *)
    InverterInputs_T01W02 : ST_MX2\Input;  (* at ECAT://node#11/d005 Multi-function Input Monitor *)
    InverterCommands_Belt_W02 : ST_MX2\Command;  (* at ECAT://node#12/Command *)
    InverterSpeed_Belt_W02 : INT;  (* at ECAT://node#12/Frequency reference *)
    InverterStatus_Belt_W02 : ST_MX2\Status;  (* at ECAT://node#12/Status *)
    InverterInputs_Belt_W02 : ST_MX2\Input;  (* at ECAT://node#12/d005 Multi-function Input Monitor *)
    Comm_T01W02_W02 : ST_FB_25050\CommInPipe;  (* Communication from T01W02 to W02 *)
    Comm_LiftGR4_W02 : ST_FB_25050\CommInPipe;  (* Communication from liftGR4 to W02 *)
    Comm_W02_T01W02 : ST_FB_25050\CommOutPipe;  (* Communication from W02 to T01W02 *)
    Comm_W02_LiftGR04 : ST_FB_25050\CommOutPipe;  (* Communication from W02 to LiftGR4 *)
END_VAR
VAR_GLOBAL RETAIN
    T01W02_Dat_A_Control AT %D20040 : ST_DatAControl_Standard;
    T01W02_Commands AT %D20057 : ST_FB_30051_Commands;
    T01W02_Direction AT %D20079 : UINT;
END_VAR
VAR_GLOBAL
    EMB_CP : BOOL;  (* Emergency stop button CP OK; at ECAT://node#[1,2]/Standard Input 1st Word/Si00 Logical Value *)
    EMB_LiftGR4 : BOOL;  (* Emergency stop button LiftGR04 OK; at ECAT://node#[8,4]/Standard Input 1st Word/Si00 Logical Value *)
    EMB_LiftGR03 : BOOL;  (* Emergency stop button LiftGR03 OK; at ECAT://node#[5,4]/Standard Input 1st Word/Si00 Logical Value *)
END_VAR
VAR_GLOBAL RETAIN
    CP AT %D20080 : ST_CP;  (* Alarm00 Alarm word 0; Alarm CP in Alarm; Manual CP manual; Enable CP Enable; Busy CP Busy; Emergencystop CP in emergencystop *)
    EncoderRackMM : UDINT;  (* Encoderwaarde rijden stelling in MM *)
END_VAR
VAR_GLOBAL
    Speed_Rack_MM_per_Sec : REAL;
    Speed_Rack_M_per_Sec : REAL;
    Speed_Rack_KM_per_Hour : REAL;
END_VAR
VAR_GLOBAL RETAIN
    EncoderXtrackMM : UDINT;  (* Encoderwaarde rijden X-track in MM *)
END_VAR
VAR_GLOBAL
    Speed_XTrack_MM_per_Sec : REAL;
    Speed_XTrack_M_per_Sec : REAL;
    Speed_XTrack_KM_per_Hour : REAL;
    InverterStatus_Belt_W01 : ST_MX2\Status;  (* Inverter status w01; at ECAT://node#17/Status *)
    InverterCommands_Belt_W01 : ST_MX2\Command;  (* at ECAT://node#17/Command *)
    InverterSpeed_Belt_W01 : INT;  (* at ECAT://node#17/Frequency reference *)
    InverterInputs_Belt_W01 : ST_MX2\Input;  (* at ECAT://node#17/d005 Multi-function Input Monitor *)
END_VAR
VAR_GLOBAL RETAIN
    W01_Commands AT %D20137 : ST_FB_25050\Commands;
    W01_Dat_A_Control AT %D20120 : ST_DatAControl_Standard;
END_VAR
VAR_GLOBAL
    Comm_LiftGR3_W01 : ST_FB_25050\CommInPipe;
    Comm_T01W01_W01 : ST_FB_25050\CommInPipe;
    Comm_W01_LiftGR3 : ST_FB_25050\CommOutPipe;
    Comm_W01_T01W01 : ST_FB_25050\CommOutPipe;
END_VAR
VAR_GLOBAL RETAIN
    T01W01_Dat_A_Control AT %D20160 : ST_DatAControl_Standard;
    T01W01_Commands AT %D20177 : ST_FB_30051_Commands;
    T01W01_Direction AT %D20199 : UINT;
    LiftGR03NotLoaded AT %D00005.00 : BOOL;
    LiftGR04NotLoaded AT %D00005.01 : BOOL;
END_VAR
VAR_GLOBAL
    N045I0100 : BOOL;  (* Emergency stop OK *)
    N045I0101 : BOOL;  (* Limit switch turning frame down *)
    N045I0102 : BOOL;  (* Limit switch turning frame middle *)
    N045I0103 : BOOL;  (* Limit switch turning frame up *)
    N045I0104 : BOOL;  (* Limit switch sprayboom left *)
    N045I0105 : BOOL;  (* Limit switch sprayboom right *)
    N045I0106 : BOOL;  (* IS container clamp 1 fixed *)
    N045I0107 : BOOL;  (* IS container clamp 1 loose *)
    N045I0108 : BOOL;  (* IS container clamp 2 fixed *)
    N045I0109 : BOOL;  (* IS container clamp 2 loose *)
    N045I0110 : BOOL;  (* Clean water level is oke *)
    N045I0111 : BOOL;  (* Level is low, start filling *)
    N045I0112 : BOOL;  (* Motor protective circuit breakers pump OK *)
    N045I0113 : BOOL;  (* IS container present on turning frame *)
    N045I0114 : BOOL;  (* IS container present on turning frame *)
    N045I0115 : BOOL;  (* Emergency stop time delayed *)
    N045O0200 : BOOL;  (* Clean water pump *)
    N045O0201 : BOOL;  (* Actuator 1 out *)
    N045O0202 : BOOL;  (* Actuator 1 In *)
    N045O0203 : BOOL;  (* Actuator 2 out *)
    N045O0204 : BOOL;  (* Actuator 2 in *)
    N045O0205 : BOOL;  (* Solenoid filling clean water reservoir *)
    N045O0206 : BOOL;  (* Solenoid clean water dirt belt *)
    N045O0207 : BOOL;  (* Lamp Red *)
    N045O0208 : BOOL;  (* Lamp Orange *)
    N045O0209 : BOOL;  (* Lamp Green *)
    N045O0210 : BOOL;  (* Brake turning frame *)
    N045O0211 : BOOL;  (* Spare output *)
    N045O0212 : BOOL;  (* Spare output *)
    N045O0213 : BOOL;  (* Spare output *)
    N045O0214 : BOOL;  (* Spare output *)
    N045O0215 : BOOL;  (* Spare output *)
    InverterCommands_W03 : ST_MX2\Command;
    InverterSpeed_W03 : INT;
    InverterOutputs_W03 : ST_MX2\Output;
    InverterStatus_W03 : ST_MX2\Status;
    InverterInputs_W03 : ST_MX2\Input;
    InverterCommands_W04 : ST_MX2\Command;
    InverterSpeed_W04 : INT;
    InverterOutputs_W04 : ST_MX2\Output;
    InverterStatus_W04 : ST_MX2\Status;
    InverterInputs_W04 : ST_MX2\Input;
    InverterCommands_W05 : ST_MX2\Command;
    InverterSpeed_W05 : INT;
    InverterOutputs_W05 : ST_MX2\Output;
    InverterStatus_W05 : ST_MX2\Status;
    InverterInputs_W05 : ST_MX2\Input;
    InverterCommands_W06 : ST_MX2\Command;  (* at ECAT://node#26/Command *)
    InverterSpeed_W06 : INT;  (* at ECAT://node#26/Frequency reference *)
    InverterOutputs_W06 : ST_MX2\Output;  (* at ECAT://node#26/Output terminal setting *)
    InverterStatus_W06 : ST_MX2\Status;  (* at ECAT://node#26/Status *)
    InverterInputs_W06 : ST_MX2\Input;  (* at ECAT://node#26/d005 Multi-function Input Monitor *)
    InverterCommands_W07 : ST_MX2\Command;  (* at ECAT://node#20/Command *)
    InverterSpeed_W07 : INT;  (* at ECAT://node#20/Frequency reference *)
    InverterOutputs_W07 : ST_MX2\Output;  (* at ECAT://node#20/Output terminal setting *)
    InverterStatus_W07 : ST_MX2\Status;  (* at ECAT://node#20/Status *)
    InverterInputs_W07 : ST_MX2\Input;  (* at ECAT://node#20/d005 Multi-function Input Monitor *)
    InverterCommands_T02W06 : ST_MX2\Command;  (* at ECAT://node#24/Command *)
    InverterSpeed_T02W06 : INT;  (* at ECAT://node#24/Frequency reference *)
    InverterStatus_T02W06 : ST_MX2\Status;  (* at ECAT://node#24/Status *)
    InverterInputs_T02W06 : ST_MX2\Input;  (* at ECAT://node#24/d005 Multi-function Input Monitor *)
    InverterCommands_T02W07 : ST_MX2\Command;  (* at ECAT://node#22/Command *)
    InverterSpeed_T02W07 : INT;  (* at ECAT://node#22/Frequency reference *)
    InverterStatus_T02W07 : ST_MX2\Status;  (* at ECAT://node#22/Status *)
    InverterInputs_T02W07 : ST_MX2\Input;  (* at ECAT://node#22/d005 Multi-function Input Monitor *)
    InverterCommands_T02_Stacker : ST_MX2\Command;  (* at ECAT://node#21/Command *)
    InverterSpeed_T02_Stacker : INT;  (* at ECAT://node#21/Frequency reference *)
    InverterStatus_T02_Stacker : ST_MX2\Status;  (* at ECAT://node#21/Status *)
    InverterInputs_T02_Stacker : ST_MX2\Input;  (* at ECAT://node#21/d005 Multi-function Input Monitor *)
    InverterCommands_Stacker : ST_MX2\Command;  (* at ECAT://node#19/Command *)
    InverterSpeed_Stacker : INT;  (* at ECAT://node#19/Frequency reference *)
    InverterOutputs_Stacker : ST_MX2\Output;  (* at ECAT://node#19/Output terminal setting *)
    InverterStatus_Stacker : ST_MX2\Status;  (* at ECAT://node#19/Status *)
    InverterInputs_Stacker : ST_MX2\Input;  (* at ECAT://node#19/d005 Multi-function Input Monitor *)
    InverterSpeed_CLE_Turn : INT;
    InverterOutputs_CLE_Turn : ST_MX2\Output;
    InverterStatus_CLE_Turn : ST_MX2\Status;
    InverterInputs_CLE_Turn : ST_MX2\Input;
    InverterCommands_CLE_Spray : ST_MX2\Command;
    InverterSpeed_CLE_Spray : INT;
    InverterOutputs_CLE_Spray : ST_MX2\Output;
    InverterStatus_CLE_Spray : ST_MX2\Status;
    InverterInputs_CLE_Spray : ST_MX2\Input;
    InverterCommands_CLE_Dirt : ST_MX2\Command;
    InverterSpeed_CLE_Dirt : INT;
    InverterOutputs_CLE_Dirt : ST_MX2\Output;
    InverterStatus_CLE_Dirt : ST_MX2\Status;
    InverterInputs_CLE_Dirt : ST_MX2\Input;
    InverterCommands_T02W07_Belt : ST_MX2\Command;  (* at ECAT://node#23/Command *)
    InverterSpeed_T02W07_Belt : INT;  (* at ECAT://node#23/Frequency reference *)
    InverterOutputs_T02W07_Belt : ST_MX2\Output;  (* at ECAT://node#23/Output terminal setting *)
    InverterStatus_T02W07_Belt : ST_MX2\Status;  (* at ECAT://node#23/Status *)
    InverterInputs_T02W07_Belt : ST_MX2\Input;  (* at ECAT://node#23/d005 Multi-function Input Monitor *)
    InverterCommands_T02W06_Belt : ST_MX2\Command;  (* at ECAT://node#25/Command *)
    InverterSpeed_T02W06_Belt : INT;  (* at ECAT://node#25/Frequency reference *)
    InverterOutputs_T02W06_Belt : ST_MX2\Output;  (* at ECAT://node#25/Output terminal setting *)
    InverterStatus_T02W06_Belt : ST_MX2\Status;  (* at ECAT://node#25/Status *)
    InverterInputs_T02W06_Belt : ST_MX2\Input;  (* at ECAT://node#25/d005 Multi-function Input Monitor *)
    Comm_T02W06_W06 : ST_FB_25050\CommInPipe;  (* Communication from T02W06 to W06 *)
    Comm_LiftGR3_W06 : ST_FB_25050\CommInPipe;  (* Communication from lift GR03 to W06 *)
    Comm_W06_T02W06 : ST_FB_25050\CommOutPipe;  (* Communication from W06 to T02W06 *)
    Comm_W06_LiftGR3 : ST_FB_25050\CommOutPipe;  (* Communication from W06 to LiftGR3 *)
    Comm_W07_T02W07 : ST_FB_25050\CommOutPipe;  (* Communication from W07 to T02W07 *)
    Comm_W07_LiftGR04 : ST_FB_25050\CommOutPipe;  (* Communication from W07 to LiftGR04 *)
END_VAR
VAR_GLOBAL RETAIN
    W07_Dat_A_Control AT %D20360 : ST_DatAControl_Standard;  (* Dat a control interface *)
    W07_Commands AT %D20377 : ST_FB_25050\Commands;  (* Comands W07 *)
END_VAR
VAR_GLOBAL
    Comm_LiftGR4_W07 : ST_FB_25050\CommInPipe;  (* Communication from lift GR04 to W07 *)
    Comm_T02W07_W07 : ST_FB_25050\CommInPipe;  (* Communication from T02W07 to W07 *)
END_VAR
VAR_GLOBAL RETAIN
    W06_Dat_A_Control AT %D20320 : ST_DatAControl_Standard;  (* Dat a control interface *)
    W06_Commands AT %D20337 : ST_FB_25050\Commands;  (* Commands W06 *)
    T02W07_DatAControl AT %D20440 : ST_DatAControl_Standard;  (* Dat a Control interface *)
    T02W07_Commands AT %D20457 : ST_FB_30051_Commands;  (* Commands T02W07 *)
    T02W06_DatAControl AT %D20400 : ST_DatAControl_Standard;  (* Datacontrol interface *)
    T02W06_Commands AT %D20417 : ST_FB_30051_Commands;  (* Commands T02W06 *)
    Stacker_DatAControl AT %D20480 : ST_DatAControl_Standard;
    Stacker_Commands AT %D20497 : ST_Stacker_Commands;
END_VAR
VAR_GLOBAL
    EMB_T01W01 : BOOL;  (* Emergency stop button OK T01W01; at ECAT://node#[1,2]/Standard Input 1st Word/Si02 Logical Value *)
    EMB_T01W02 : BOOL;  (* Emergency stop button OK T01W02; at ECAT://node#[1,2]/Standard Input 1st Word/Si03 Logical Value *)
    EMB_T02W06 : BOOL;  (* Emergency stop button OK T02W06; at ECAT://node#[1,2]/Standard Input 1st Word/Si05 Logical Value *)
    EMB_T02W07 : BOOL;  (* Emergency stop button OK T02W07; at ECAT://node#[1,2]/Standard Input 1st Word/Si06 Logical Value *)
    EMB_ATC : BOOL;  (* Emergency stop button OK ATC Desk; at ECAT://node#[1,2]/Standard Input 1st Word/Si07 Logical Value *)
    InverterCommands_CLE_Turn : ST_MX2\Command;
END_VAR
VAR_GLOBAL RETAIN
    Cleaner_Commands AT %D20537 : ST_FB_40303_Commands;  (* Commands Cleaner *)
    Comm_To_Carrier03 AT %D06000 : ST_FB_40701\Comm_IN;  (* ST Comm from Carrier03 *)
    Comm_To_Carrier03_SENDREC AT %D06000 : ARRAY[0..199] OF WORD;  (* Comm from Carrier02 (For send/recieve) *)
    GrantEnter_Ca03 AT %D00993.00 : BOOL;  (* Grant Enter carrier03 self *)
    GrantLeave_Ca03 AT %D00993.01 : BOOL;  (* Grant Leave carrier03 self *)
    Comm_From_Carrier03 AT %D06200 : ST_FB_40701\Comm_OUT;  (* ST Comm from Carrier03 *)
END_VAR
VAR_GLOBAL
    CommSend_Ca03 : BOOL;  (* Communication send to Carrier03 *)
    CommReceive_Ca03 : BOOL;  (* Communication receive from Carrier03 *)
    DstNetAdr_Ca03 : _sDNET_ADR;  (* Send adress Carrier03 *)
    Option_Ca03 : _sRESPONSE;  (* Send options Carrier03 *)
    Comm_LiftGR4_W03 : ST_FB_25050\CommInPipe;  (* Communication from lift GR04 to W03 *)
    Comm_LiftGR4_W05 : ST_FB_25050\CommInPipe;  (* Communication from lift GR04 to W05 *)
    Comm_W03_LiftGR04 : ST_FB_25050\CommOutPipe;  (* Communication from W03 to LiftGR4 *)
    Comm_W05_LiftGR04 : ST_FB_25050\CommOutPipe;  (* Communication from W05 to LiftGR4 *)
    Comm_W03_W04 : ST_FB_25050\CommInPipe;  (* Communication from W03 tot W04 *)
    Comm_W04_W03 : ST_FB_25050\CommInPipe;  (* Communication from W04 tot W03 *)
    Comm_W05_W04 : ST_FB_25050\CommInPipe;  (* Communication from W05 tot W04 *)
    Comm_W04_W05 : ST_FB_25050\CommInPipe;  (* Communication from W04 tot W05 *)
END_VAR
VAR_GLOBAL RETAIN
    T02W07_Direction AT %D20479 : UINT;
    T02W06_Direction AT %D20439 : UINT;
END_VAR
VAR_GLOBAL
    Comm_T01_T01W01 : ST_FB_30051_CommIn202;  (* Communication rom T01 to T01W01 *)
    Comm_T01_T01W02 : ST_FB_30051_CommIn201;  (* Communication rom T01 to T01W02 *)
END_VAR
VAR_GLOBAL RETAIN
    EncoderLift03 AT %D22020 : UDINT;  (* Current encoder value of lift 03 *)
    EncoderLift04 AT %D22050 : UDINT;  (* Current encoder value of lift 04 *)
    Lift3_PulsValueLevel1 AT %D22022 : UDINT;
    Lift3_PulsValueLevel2 AT %D22024 : UDINT;
    Lift3_PulsValueLevel3 AT %D22026 : UDINT;
    Lift3_PulsValueLevel4 AT %D22028 : UDINT;
    Lift3_PulsValueLevel5 AT %D22030 : UDINT;
    Lift3_PulsValueLevel6 AT %D22032 : UDINT;
    Lift3_PulsValueLevel7 AT %D22034 : UDINT;
    Lift3_PulsValueLevel8 AT %D22036 : UDINT;
    Lift3_PulsValueLevel9 AT %D22038 : UDINT;
    Lift4_PulsValueLevel1 AT %D22052 : UDINT;
    Lift4_PulsValueLevel2 AT %D22054 : UDINT;
    Lift4_PulsValueLevel3 AT %D22056 : UDINT;
    Lift4_PulsValueLevel4 AT %D22058 : UDINT;
    Lift4_PulsValueLevel5 AT %D22060 : UDINT;
    Lift4_PulsValueLevel6 AT %D22062 : UDINT;
    Lift4_PulsValueLevel7 AT %D22064 : UDINT;
    Lift4_PulsValueLevel8 AT %D22066 : UDINT;
    Lift4_PulsValueLevel9 AT %D22068 : UDINT;
    Lift4_PulsValueLevel10 AT %D22070 : UDINT;
    Lift3_PulsValueLevel1_Backup AT %D22122 : UDINT;
    Lift3_PulsValueLevel2_Backup AT %D22124 : UDINT;
    Lift3_PulsValueLevel3_Backup AT %D22126 : UDINT;
    Lift3_PulsValueLevel4_Backup AT %D22128 : UDINT;
    Lift3_PulsValueLevel5_Backup AT %D22130 : UDINT;
    Lift3_PulsValueLevel6_Backup AT %D22132 : UDINT;
    Lift3_PulsValueLevel7_Backup AT %D22134 : UDINT;
    Lift3_PulsValueLevel8_Backup AT %D22136 : UDINT;
    Lift3_PulsValueLevel9_Backup AT %D22138 : UDINT;
    Lift4_PulsValueLevel1_Backup AT %D22152 : UDINT;
    Lift4_PulsValueLevel2_Backup AT %D22154 : UDINT;
    Lift4_PulsValueLevel3_Backup AT %D22156 : UDINT;
    Lift4_PulsValueLevel4_Backup AT %D22158 : UDINT;
    Lift4_PulsValueLevel5_Backup AT %D22160 : UDINT;
    Lift4_PulsValueLevel6_Backup AT %D22162 : UDINT;
    Lift4_PulsValueLevel7_Backup AT %D22164 : UDINT;
    Lift4_PulsValueLevel8_Backup AT %D22166 : UDINT;
    Lift4_PulsValueLevel9_Backup AT %D22168 : UDINT;
    Lift4_PulsValueLevel10_Backup AT %D22170 : UDINT;
END_VAR
VAR_GLOBAL
    N000O0103 : BOOL;  (* Charger_3D202; at ECAT://node#[1,1]/Output Bit 16 bits/Output Bit 03 *)
    N000O0104 : BOOL;  (* at ECAT://node#[1,1]/Output Bit 16 bits/Output Bit 04 *)
    N000O0105 : BOOL;  (* at ECAT://node#[1,1]/Output Bit 16 bits/Output Bit 05 *)
END_VAR
VAR_GLOBAL RETAIN
    Lift3_Extra_Warning1 AT %D23020 : WORD;
    Lift3_Extra_Warning2 AT %D23021 : WORD;
    Lift4_Extra_Warning1 AT %D23050 : WORD;
    Lift4_Extra_Warning2 AT %D23051 : WORD;
    LC_Lift3_Disable_Front_Level7 AT %D00007.09 : BOOL;
    LC_LIft4_Disable_Back_Level0 AT %D00008.00 : BOOL;
    LC_LIft4_Disable_Back_Level4 AT %D00008.01 : BOOL;
    LC_LIft4_Disable_Front_Level0 AT %D00008.02 : BOOL;
    LC_LIft4_Disable_Front_Level1 AT %D00008.03 : BOOL;
    LC_LIft4_Disable_Front_Level2 AT %D00008.04 : BOOL;
    LC_LIft4_Disable_Front_Level3 AT %D00008.05 : BOOL;
    LC_LIft4_Disable_Front_Level4 AT %D00008.06 : BOOL;
    LC_LIft4_Disable_Front_Level5 AT %D00008.07 : BOOL;
    LC_LIft4_Disable_Front_Level6 AT %D00008.08 : BOOL;
    LC_LIft4_Disable_Front_Level7 AT %D00008.09 : BOOL;
    Lift4_Extra_Warning3 AT %D23052 : WORD;
    Lift3_Extra_Warning3 AT %D23022 : WORD;
    WarningBadCommC1 AT %D00005.08 : BOOL;  (* Warning bad comm carrier 1 *)
    WarningBadCommC2 AT %D00005.09 : BOOL;  (* Warning bad comm carrier 2 *)
    WarningBadCommC3 AT %D00005.10 : BOOL;  (* Warning bad comm carrier 3 *)
    Comm_From_Carrier04 AT %D06600 : ST_FB_40701\Comm_OUT;  (* ST Comm from Carrier04 *)
END_VAR
VAR_GLOBAL
    Option_Ca04 : _sRESPONSE;  (* Send options Carrier04 *)
    DstNetAdr_Ca04 : _sDNET_ADR;  (* Send adress Carrier04 *)
    CommSend_Ca04 : BOOL;  (* Communication send to Carrier04 *)
    CommReceive_Ca04 : BOOL;  (* Communication receive from Carrier04 *)
END_VAR
VAR_GLOBAL RETAIN
    RegistrationData_Carrier04 AT %D07600 : ARRAY[0..199] OF UINT;  (* Registration data *)
    GrantEnter_Ca04 AT %D00994.00 : BOOL;  (* Grant Enter carrier04 self *)
    GrantLeave_Ca04 AT %D00994.01 : BOOL;  (* Grant Leave carrier04 self *)
    Comm_To_Carrier05_SENDREC AT %D08000 : ARRAY[0..199] OF WORD;  (* Comm from Carrier05 (For send/recieve) *)
    Comm_To_Carrier05 AT %D08000 : ST_FB_40701\Comm_IN;  (* ST Comm from Carrier05 *)
    Comm_From_Carrier05_SENDREC AT %D08200 : ARRAY[0..199] OF WORD;  (* Comm from Carrier05 (For send/recieve) *)
    Comm_From_Carrier05 AT %D08200 : ST_FB_40701\Comm_OUT;  (* ST Comm from Carrier05 *)
END_VAR
VAR_GLOBAL
    Option_Ca05 : _sRESPONSE;  (* Send options Carrier05 *)
    DstNetAdr_Ca05 : _sDNET_ADR;  (* Send adress Carrier05 *)
    CommSend_Ca05 : BOOL;  (* Communication send to Carrier05 *)
    CommReceive_Ca05 : BOOL;  (* Communication receive from Carrier05 *)
END_VAR
VAR_GLOBAL RETAIN
    RegistrationData_Carrier05 AT %D07800 : ARRAY[0..199] OF UINT;  (* Registration data *)
    GrantEnter_Ca05 AT %D00995.00 : BOOL;  (* Grant Enter carrier05self *)
    GrantLeave_Ca05 AT %D00995.01 : BOOL;  (* Grant Leave carrier05 self *)
    WarningBadCommC4 AT %D00005.11 : BOOL;  (* Warning bad comm carrier 4 *)
    WarningBadCommC5 AT %D00005.12 : BOOL;  (* Warning bad comm carrier 5 *)
END_VAR
VAR_GLOBAL
    Error_Status_N43 : BYTE;
    Error_Status_N8 : BYTE;
    Error_Status_N33 : BYTE;
    Error_Status_N5 : BYTE;
    N08_Minor_Fault : BOOL;  (* at ECAT://node#8/Sysmac Error Status/Minor Fault *)
    N08_Partial_Fault : BOOL;  (* at ECAT://node#8/Sysmac Error Status/Partial Fault *)
    N08_Major_Fault : BOOL;  (* at ECAT://node#8/Sysmac Error Status/Major Fault *)
    N43_Minor_Fault : BOOL;  (* at ECAT://node#43/Sysmac Error Status/Minor Fault *)
    N43_Partial_Fault : BOOL;  (* at ECAT://node#43/Sysmac Error Status/Partial Fault *)
    N43_Major_Fault : BOOL;  (* at ECAT://node#43/Sysmac Error Status/Major Fault *)
    N05_Minor_Fault : BOOL;  (* at ECAT://node#5/Sysmac Error Status/Minor Fault *)
    N05_Partial_Fault : BOOL;  (* at ECAT://node#5/Sysmac Error Status/Partial Fault *)
    N05_Major_Fault : BOOL;  (* at ECAT://node#5/Sysmac Error Status/Major Fault *)
    N33_Minor_Fault : BOOL;  (* at ECAT://node#33/Sysmac Error Status/Minor Fault *)
    N33_Partial_Fault : BOOL;  (* at ECAT://node#33/Sysmac Error Status/Partial Fault *)
    N33_Major_Fault : BOOL;  (* at ECAT://node#33/Sysmac Error Status/Major Fault *)
END_VAR
VAR_GLOBAL RETAIN
    Lift03_Status AT %D23023 : ST_FB_40401_Status;
    Lift04_Status AT %D23053 : ST_FB_40401_Status;
    Charger4D105_DatAControl AT %D20680 : ST_DatAControl_Standard;
    Commands_Charger4D105 AT %D20697 : ST_FB_1xxxx\FB_10001_Commands;
    Commands_Charger3D105 AT %D20737 : ST_FB_1xxxx\FB_10001_Commands;
    Charger3D105_DatAControl AT %D20720 : ST_DatAControl_Standard;
    Charger4D402_DatAControl AT %D20560 : ST_DatAControl_Standard;
    Commands_Charger4D402 AT %D20577 : ST_FB_1xxxx\FB_10001_Commands;
    Charger4D102_DatAControl AT %D20600 : ST_DatAControl_Standard;
    Commands_Charger4D102 AT %D20617 : ST_FB_1xxxx\FB_10001_Commands;
    Charger3D202_DatAControl AT %D20640 : ST_DatAControl_Standard;
    Commands_Charger3D202 AT %D20657 : ST_FB_1xxxx\FB_10001_Commands;
    LC_Lift3_Disable_Front_Level6 AT %D00007.08 : BOOL;
    T02W07_Loaded AT %D00006.05 : BOOL;
END_VAR

(* Program Program0: safety or other program stored in binary form, left out *)

PROGRAM General
VAR
    T_Power_OK : _sTimer;  (* Timer power up on PLC OK *)
    Manual_ReadSettings : BOOL;  (* Write settings by activating the script manually *)
    CommCounter : UINT;  (* Running Timer Communications *)
    EthercatErrorLevel : UINT;
    EthercatErrorCode : DWORD;
    CP_ResetAlrm : BOOL;  (* reset alarm *)
    ResetErrorEthercat : ResetECError;
    ResetErrorPLC : ResetPLCError;
END_VAR
VAR_EXTERNAL
    I_EStop_OK : BOOL;
    ES_OK : BOOL;  (* Emergencystop OK *)
    Trig_ReadSettings : BOOL;
    SafetyRelays_Lift03 : BOOL;
    SafetyRelays_Lift04 : BOOL;
    Led_RS_Extern : BOOL;
    TransferBuffer : ST_TransferBuffer;  (* TransferBuffer *)
    CommSend_Ca01 : BOOL;  (* Communication send to Carrier01 *)
    CommReceive_Ca01 : BOOL;
    CommSend_Ca02 : BOOL;
    CommReceive_Ca02 : BOOL;
    Transfer_BenchSize : UINT;  (* Size of bench to be moved. *)
    N000O0102 : BOOL;
    EMB_CP : BOOL;
    Dummy : BOOL;
    EMB_LiftGR4 : BOOL;
    EMB_LiftGR03 : BOOL;
    CP : ST_CP;  (* Alarm00 Alarm word 0; Alarm CP in Alarm; Manual CP manual; Enable CP Enable; Busy CP Busy; Emergencystop CP in emergencystop; Alarm01 Alarm word 1 *)
    EMB_T01W01 : BOOL;
    EMB_T01W02 : BOOL;
    EMB_T02W06 : BOOL;
    EMB_T02W07 : BOOL;
    CommSend_Ca03 : BOOL;
    CommReceive_Ca03 : BOOL;
    EMB_ATC : BOOL;
    CommSend_Ca04 : BOOL;
    CommReceive_Ca04 : BOOL;
    CommSend_Ca05 : BOOL;
    CommReceive_Ca05 : BOOL;
END_VAR
VAR
    _t1 : BOOL;
    _e2 : R_TRIG;
    _e3 : R_TRIG;
    _t4 : BOOL;
    _e5 : R_TRIG;
END_VAR

(* Section EStop: ladder, written here as Structured Text *)

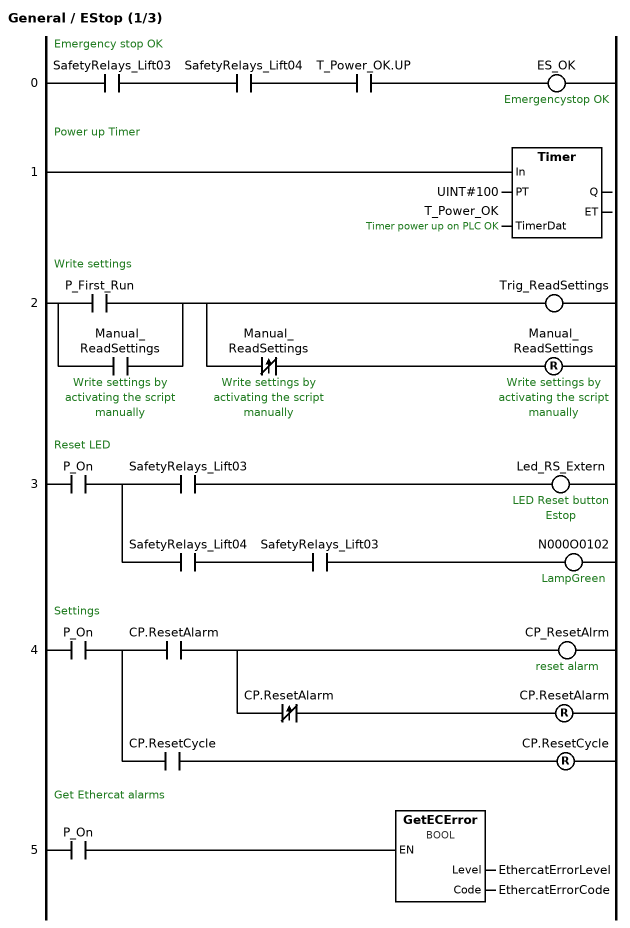
(* Rung 0: Emergency stop OK *)
ES_OK := SafetyRelays_Lift03 AND SafetyRelays_Lift04 AND T_Power_OK.UP;
(* Rung 1: Power up Timer *)
_t1 := Timer(In := TRUE, PT := UINT#100, TimerDat := T_Power_OK);
(* Rung 2: Write settings *)
Trig_ReadSettings := P_First_Run OR Manual_ReadSettings;
_e2(CLK := Manual_ReadSettings);
IF (P_First_Run OR Manual_ReadSettings) AND NOT _e2.Q THEN Manual_ReadSettings := FALSE; END_IF;
(* Rung 3: Reset LED *)
Led_RS_Extern := P_On AND SafetyRelays_Lift03;
N000O0102 := P_On AND SafetyRelays_Lift04 AND SafetyRelays_Lift03;
(* Rung 4: Settings *)
CP_ResetAlrm := P_On AND CP.ResetAlarm;
_e3(CLK := CP.ResetAlarm);
IF P_On AND CP.ResetAlarm AND NOT _e3.Q THEN CP.ResetAlarm := FALSE; END_IF;
IF P_On AND CP.ResetCycle THEN CP.ResetCycle := FALSE; END_IF;
(* Rung 5: Get Ethercat alarms *)
_t4 := FALSE;
IF P_On THEN _t4 := GetECError(Level => EthercatErrorLevel, Code => EthercatErrorCode); END_IF;

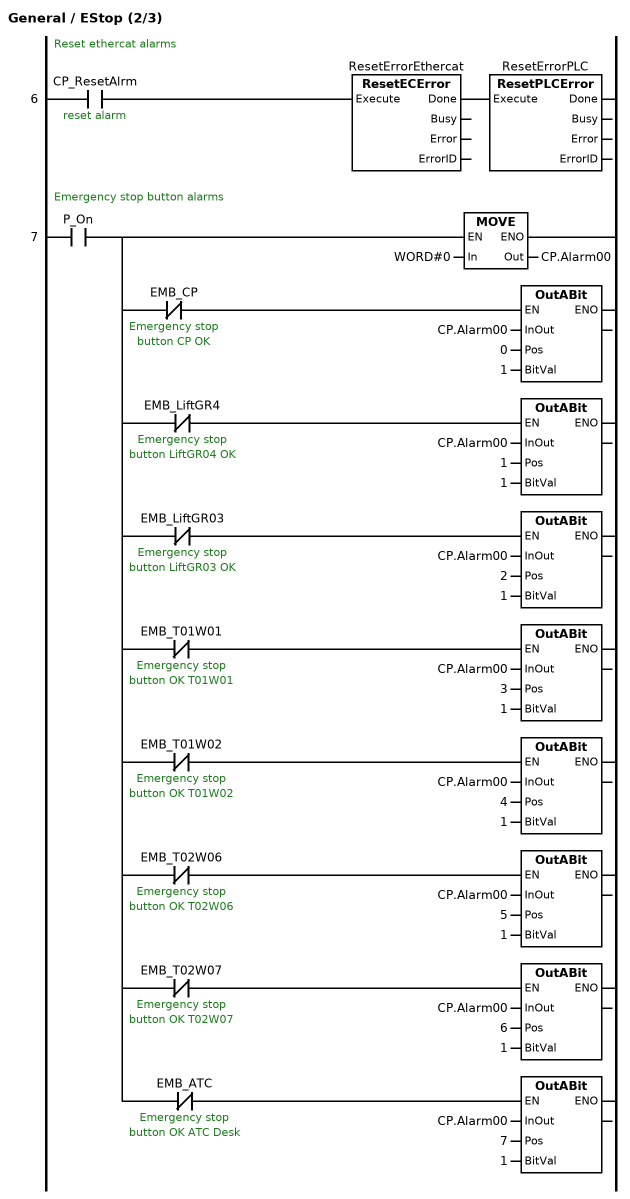
(* Rung 6: Reset ethercat alarms *)
ResetErrorEthercat(Execute := CP_ResetAlrm);
ResetErrorPLC(Execute := ResetErrorEthercat.Done);
(* Rung 7: Emergency stop button alarms *)
IF P_On THEN CP.Alarm00 := WORD#0; END_IF;
IF P_On AND NOT EMB_CP THEN OutABit(InOut := CP.Alarm00, Pos := 0, BitVal := 1); END_IF;
IF P_On AND NOT EMB_LiftGR4 THEN OutABit(InOut := CP.Alarm00, Pos := 1, BitVal := 1); END_IF;
IF P_On AND NOT EMB_LiftGR03 THEN OutABit(InOut := CP.Alarm00, Pos := 2, BitVal := 1); END_IF;
IF P_On AND NOT EMB_T01W01 THEN OutABit(InOut := CP.Alarm00, Pos := 3, BitVal := 1); END_IF;
IF P_On AND NOT EMB_T01W02 THEN OutABit(InOut := CP.Alarm00, Pos := 4, BitVal := 1); END_IF;
IF P_On AND NOT EMB_T02W06 THEN OutABit(InOut := CP.Alarm00, Pos := 5, BitVal := 1); END_IF;
IF P_On AND NOT EMB_T02W07 THEN OutABit(InOut := CP.Alarm00, Pos := 6, BitVal := 1); END_IF;
IF P_On AND NOT EMB_ATC THEN OutABit(InOut := CP.Alarm00, Pos := 7, BitVal := 1); END_IF;

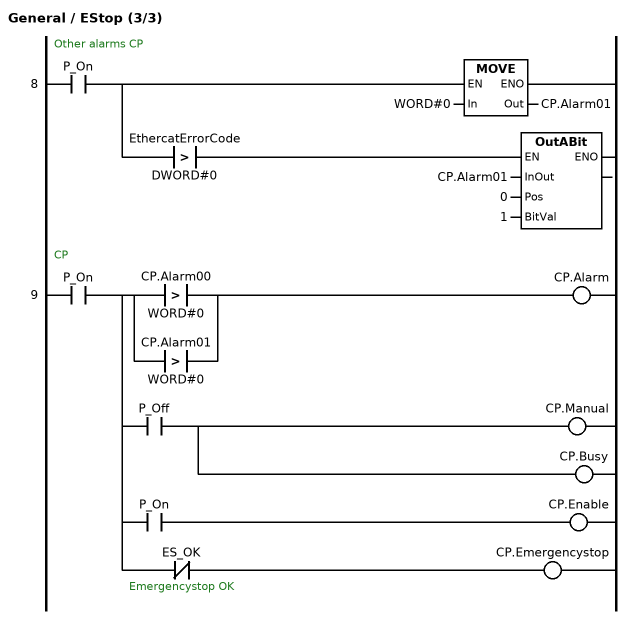
(* Rung 8: Other alarms CP *)
IF P_On THEN CP.Alarm01 := WORD#0; END_IF;
IF P_On AND (EthercatErrorCode > DWORD#0) THEN
    OutABit(InOut := CP.Alarm01, Pos := 0, BitVal := 1);
END_IF;
(* Rung 9: CP *)
CP.Alarm := P_On AND ((CP.Alarm00 > WORD#0) OR (CP.Alarm01 > WORD#0));
CP.Manual := P_On AND P_Off;
CP.Busy := P_On AND P_Off;
CP.Enable := P_On AND P_On;
CP.Emergencystop := P_On AND NOT ES_OK;

(* Section Dat_A_Control: ladder, written here as Structured Text *)

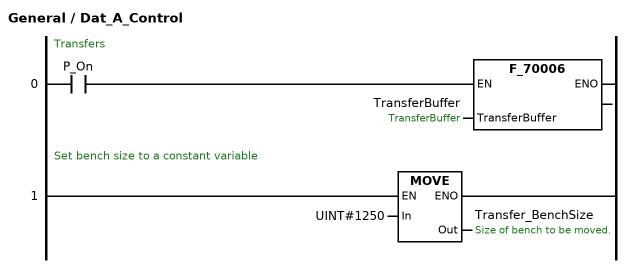
(* Rung 0: Transfers *)
IF P_On THEN F_70006(TransferBuffer := TransferBuffer); END_IF;
(* Rung 1: Set bench size to a constant variable *)
Transfer_BenchSize := UINT#1250;

(* Section Communications: ladder, written here as Structured Text *)

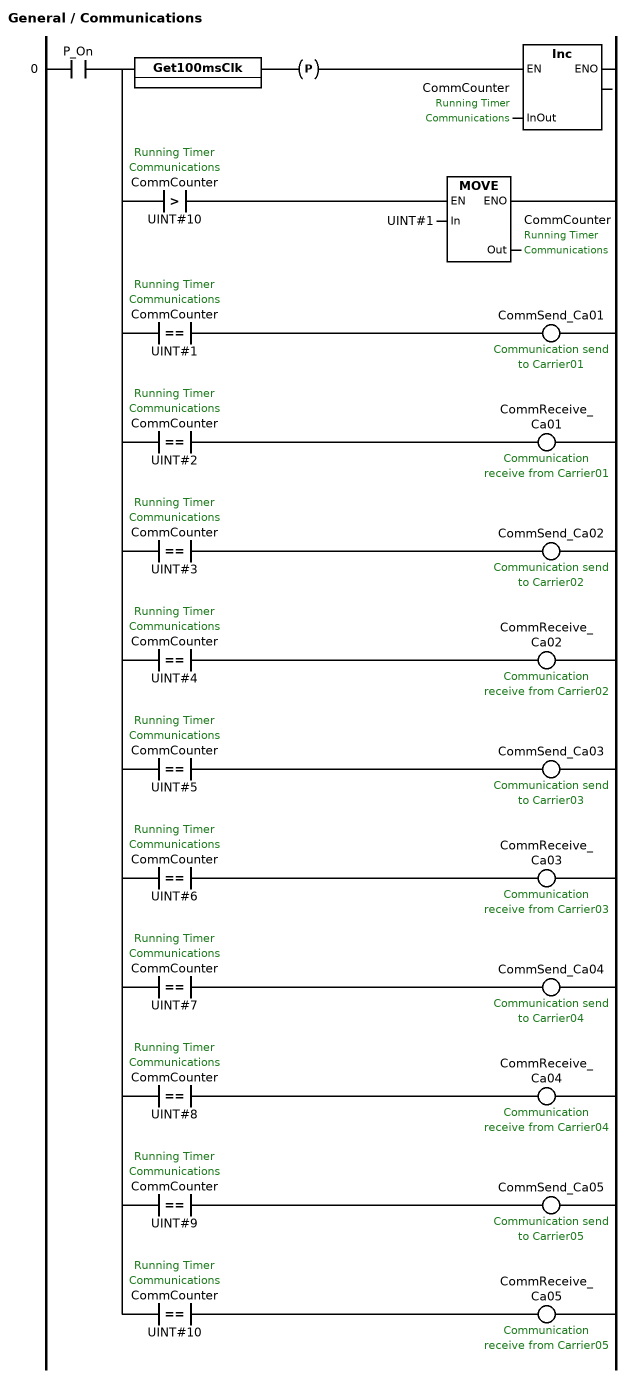
(* Rung 0 *)
_e5(CLK := P_On AND Get100msClk());
IF _e5.Q THEN Inc(InOut := CommCounter); END_IF;
IF P_On AND (CommCounter > UINT#10) THEN CommCounter := UINT#1; END_IF;
CommSend_Ca01 := P_On AND (CommCounter = UINT#1);
CommReceive_Ca01 := P_On AND (CommCounter = UINT#2);
CommSend_Ca02 := P_On AND (CommCounter = UINT#3);
CommReceive_Ca02 := P_On AND (CommCounter = UINT#4);
CommSend_Ca03 := P_On AND (CommCounter = UINT#5);
CommReceive_Ca03 := P_On AND (CommCounter = UINT#6);
CommSend_Ca04 := P_On AND (CommCounter = UINT#7);
CommReceive_Ca04 := P_On AND (CommCounter = UINT#8);
CommSend_Ca05 := P_On AND (CommCounter = UINT#9);
CommReceive_Ca05 := P_On AND (CommCounter = UINT#10);
END_PROGRAM

PROGRAM Mobile_Machines
VAR
    Lift03_WP : BOOL;
    Lift03_WPD : BOOL;
    Lift03_RV : BOOL;
    Lift03_FW : BOOL;
    Lift03_Speed : INT;
    Lift03_Reset : BOOL;
    Lift03_Alarms : BYTE;
    Knop_FW_Lift03 : BOOL;
    Knop_RV_Lift03 : BOOL;
    Knop_OK_Lift03 : BOOL;
    Knop_Snel_Lift03 : BOOL;
    Lift03_LS_Up : BOOL;
    Lift03_LS_Down : BOOL;
    Lift03_LS_FallProtect : BOOL;
    Lift03_Parameters : ST_MX2\Parameters;
    Lift03_MINSpeed : INT;
    Lift03_MAXSpeed : INT;
    Lift03_SpeedReleaseBrakes : UINT;
    Lift03_NodeNumber : UINT;
    Lift03_SafetyInput1 : BOOL;
    Lift03_SafetyInput2 : BOOL;
    Lift03_Vrijgave : BOOL;
    Led_Knop_OK_Lift03 : BOOL;
    Lift04_WP : BOOL;
    Lift04_WPD : BOOL;
    Lift04_RV : BOOL;
    Lift04_FW : BOOL;
    Lift04_Speed : INT;
    Lift04_Reset : BOOL;
    Lift04_Alarms : BYTE;
    Lift04_Alarms_Ch : BYTE;
    Knop_FW_Lift04 : BOOL;
    Knop_RV_Lift04 : BOOL;
    Knop_OK_Lift04 : BOOL;
    Knop_Snel_Lift04 : BOOL;
    Lift04_LS_Up : BOOL;
    Lift04_LS_Down : BOOL;
    Lift04_LS_FallProtect : BOOL;
    Lift04_Parameters : ST_MX2\Parameters;
    Lift04_MINSpeed : INT;
    Lift04_MAXSpeed : INT;
    Lift04_SpeedReleaseBrakes : UINT;
    Lift04_NodeNumber : UINT;
    Lift04_SafetyInput1 : BOOL;
    Lift04_SafetyInput2 : BOOL;
    Lift03_NodeNumber_Ch : UINT;
    Lift03_Speed_Ch : INT;
    Lift03_Reset_Ch : BOOL;
    Lift03_Parameters_Ch : ST_MX2\Parameters;
    Lift03_WP_Ch : BOOL;
    Lift03_WPD_Ch : BOOL;
    Lift03_Alarms_Ch : BYTE;
    Lift03_FW_Ch : BOOL;
    Lift03_RV_Ch : BOOL;
    Lift04_NodeNumber_Ch : UINT;
    Lift04_Speed_Ch : INT;
    Lift04_Reset_Ch : BOOL;
    Lift04_Parameters_Ch : ST_MX2\Parameters;
    Lift04_WP_Ch : BOOL;
    Lift04_WPD_Ch : BOOL;
    Lift04_FW_Ch : BOOL;
    Lift04_RV_Ch : BOOL;
    SettingsLift03 : ST_FB_40401_SettingsLift;  (* Settings Lift 03 *)
    SettingsLift04 : ST_FB_40401_SettingsLift;  (* Settings Lift 04 *)
    InputsLift03 : ST_FB_40401_InputsLift;
    InputsLift04 : ST_FB_40401_InputsLift;
    OutputsLift03 : ST_FB_40401_OutputsLift;
    OutputsLift04 : ST_FB_40401_OutputsLift;
    ResetEncoderValue_Lift03 : UDINT;  (* Reset encoder value of lift 03 at position *)
    ResetEncoderValue_Lift04 : UDINT;  (* Reset encoder value of lift 04 at position *)
END_VAR
VAR RETAIN
    EncoderLift03_Backup : UDINT;  (* Backup enocder value of lift 03 *)
    EncoderLift04_Backup : UDINT;  (* Backup enocder value of lift 04 *)
END_VAR
VAR
    PresetDone_Lift03 : BOOL;  (* Preset encoder lift 03 at power up *)
    PresetDone_Lift04 : BOOL;  (* Preset encoder lift 04 at power up *)
    ResetEncoder_Lift03 : BOOL;  (* Reset encoder lift 03 when at position *)
    ResetEncoder_Lift04 : BOOL;  (* Reset encoder lift 04 when at position *)
    Comm_CarX_Lift03 : ST_Comm_MobileMachine_To_Lift;  (* Communication CarrierX to Lift03 *)
    Lift03Reset_Ch : BOOL;
    Led_Knop_OK_Lift04 : BOOL;
    Lift04_Vrijgave : BOOL;
    Lift_03 : FB_40401;
    Lift_04 : FB_40401;
    Comm_Lift04_CarX : ST_Comm_Lift_To_MobileMachine;
    Comm_CarX_Lift04 : ST_Comm_MobileMachine_To_Lift;  (* Communication CarrierX to Lift04 *)
    FB_Watchdog_Carrier02 : FB_304;
    FB_Watchdog_Carrier01 : FB_304;
    MatchingArea : ST_Area;  (* Matching area *)
    MatchingXTrackNumber : UINT;  (* Matching X-Track number *)
    Transfergate_Car01 : UINT;  (* Transfergate to use *)
    Transfergate_Car02 : UINT;  (* Transfergate to use *)
    Transfergate_Car03 : UINT;  (* Transfergate to use *)
    Ca1_GrantEnter_AtThisPosition : BOOL;  (* Grant Enter at this position *)
    Ca1_GrantLeave_AtThisPosition : BOOL;  (* Grant Leave at this position *)
    TransferOK : BOOL;  (* Transfer OK *)
    BusyS_Ca01 : BOOL;  (* Busy send to Carrier01 *)
    Send_Carrier_01 : Send;
    BusyR_Ca01 : BOOL;  (* Busy receive from Carrier01 *)
    Receive_Carrier_01 : Rcv;
    Send_Carrier_02 : Send;
    BusyS_Ca02 : BOOL;  (* Busy send from Carrier02 *)
    BusyR_Ca02 : BOOL;  (* Busy recieve from Carrier02 *)
    BusyS_Ca03 : BOOL;  (* Busy send from Carrier03 *)
    BusyR_Ca03 : BOOL;  (* Busy recieve from Carrier03 *)
    Ca2_GrantEnter_AtThisPosition : BOOL;  (* Grant Enter at this position *)
    Ca2_GrantLeave_AtThisPosition : BOOL;  (* Grant Leave at this position *)
    Receive_Carrier_02 : Rcv;
    test001 : BOOL;
    CommIn_Back_GR4 : ST_FB_40401_CommIn;  (* Comm in from back *)
    CommOUT_Back_GR4 : ST_FB_40401_CommOut;  (* Comm out back *)
    Comm_Lift03_CarX : ST_Comm_Lift_To_MobileMachine;
    EncoderLift04MM : UDINT;
    PulsesPerMeterLift04 : UDINT;
    Speed_Lift04_MM_per_Sec : REAL;
    Speed_Lift04_M_per_Sec : REAL;
    Speed_Lift04_KM_per_Hour : REAL;
    EncoderLift03MM : UDINT;
    PulsesPerMeterLift03 : UDINT;
    Speed_Lift03_MM_per_Sec : REAL;
    Speed_Lift03_M_per_Sec : REAL;
    Speed_Lift03_KM_per_Hour : REAL;
    DatAControl : ST_DatAControl_Standard;  (* IN.MachineMode Machine mode; IN Data control in; OUT Dat A Control out; IN.Instruction.Operand1 Operand 1; IN.Settings.ResetAlarm Reset alar *)
    SpeedLift03 : FB_308;
    SpeedLift04 : FB_308;
    ReservationInputErr_Car1 : BOOL;  (* Reservation input error carrier 1 *)
    ReservationInputErr_Car2 : BOOL;  (* Reservation input error carrier 2 *)
    ReservationInputErr_Car3 : BOOL;  (* Reservation input error carrier 3 *)
    CommIn_Back_GR03 : ST_FB_40401_CommIn;  (* Communication in back *)
    CommOut_Back_GR03 : ST_FB_40401_CommOut;  (* Communication out back *)
    temp1 : BOOL;
    Temp2 : BOOL;
    test45 : BOOL;
    Test46 : BOOL;
    Test50 : BOOL;
    TestCarrier : BOOL;
    TestPallet : BOOL;
    test41 : BOOL;
    FB_Watchdog_Carrier03 : FB_304;
    Ca3_GrantEnter_AtThisPosition : BOOL;  (* Grant Enter at this position *)
    Ca3_GrantLeave_AtThisPosition : BOOL;  (* Grant Leave at this position *)
    Send_Carrier_03 : Send;
    Receive_Carrier_03 : Rcv;
    CommOut_Front_GR4 : ST_FB_40401_CommOut;  (* Comm out front *)
    CommIn_Front_GR4 : ST_FB_40401_CommIn;  (* Comm in front *)
    CommOut_Front_GR3 : ST_FB_40401_CommOut;  (* Comm out front *)
    CommIn_Front_GR3 : ST_FB_40401_CommIn;  (* Comm in front *)
    Carrier1_Request_Comm_Lift3 : BOOL;
    Carrier2_Request_Comm_Lift3 : BOOL;
    Carrier3_Request_Comm_Lift3 : BOOL;
    Carrier1_Request_Comm_Lift4 : BOOL;
    Carrier2_Request_Comm_Lift4 : BOOL;
    Carrier3_Request_Comm_Lift4 : BOOL;
    Manual_Backup_EncoderGR03 : BOOL;
    Manual_Backup_EncoderGR04 : BOOL;
    MoveFast_Lift03 : BOOL;
    MoveFast_Lift04 : BOOL;
    ReleasBrakeFront : BOOL;
    UserSettingsLift3 : ST_FB_40401_UserSetting;  (* User settings lift 3 *)
    UserSettingsLift4 : ST_FB_40401_UserSetting;  (* User settings lift 4 *)
    TimerbadComm_C1 : _sTimer;  (* Timer bad communication *)
    TimerbadComm_C2 : _sTimer;  (* Timer bad communication *)
    TimerbadComm_C3 : _sTimer;  (* Timer bad communication *)
    Carrier1_OutOfSystem : BOOL;  (* Carrier 1 is out of system *)
    Carrier3_OutOfSystem : BOOL;  (* Carrier 3 is out of system *)
    Carrier2_OutOfSystem : BOOL;  (* Carrier 2 is out of system *)
    FB_Watchdog_Carrier04 : FB_304;
    TimerbadComm_C4 : _sTimer;  (* Timer bad communication *)
    Carrier4_OutOfSystem : BOOL;  (* Carrier 4 is out of system *)
    Transfergate_Car04 : UINT;  (* Transfergate to use *)
    Ca4_GrantEnter_AtThisPosition : BOOL;  (* Grant Enter at this position *)
    Ca4_GrantLeave_AtThisPosition : BOOL;  (* Grant Leave at this position *)
    ReservationInputErr_Car4 : BOOL;  (* Reservation input error carrier 4 *)
    BusyS_Ca04 : BOOL;  (* Busy send from Carrier04 *)
    Send_Carrier_04 : Send;
    BusyR_Ca04 : BOOL;  (* Busy recieve from Carrier04 *)
    Receive_Carrier_04 : Rcv;
    FB_Watchdog_Carrier05 : FB_304;
    TimerbadComm_C5 : _sTimer;  (* Timer bad communication *)
    Carrier5_OutOfSystem : BOOL;  (* Carrier 5 is out of system *)
    Transfergate_Car05 : UINT;  (* Transfergate to use *)
    Ca5_GrantEnter_AtThisPosition : BOOL;  (* Grant Enter at this position *)
    Ca5_GrantLeave_AtThisPosition : BOOL;  (* Grant Leave at this position *)
    ReservationInputErr_Car5 : BOOL;  (* Reservation input error carrier 5 *)
    BusyS_Ca05 : BOOL;  (* Busy send from Carrier05 *)
    Send_Carrier_05 : Send;
    BusyR_Ca05 : BOOL;  (* Busy recieve from Carrier05 *)
    Receive_Carrier_05 : Rcv;
    StartCharger_4D402 : BOOL;
    StartCharger_4D102 : BOOL;
    StartCharger_3D202 : BOOL;
    StartCharger_4D105 : BOOL;
    StartCharger_3D105 : BOOL;
    FB_Charger4D105 : FB_10001;
    FB_Charger3D105 : FB_10001;
    FB_Charger4D402 : FB_10001;
    FB_Charger4D102 : FB_10001;
    FB_Charger3D202 : FB_10001;
END_VAR
VAR_EXTERNAL
    Freq_Lift04 : UINT;
    N005I0200 : BOOL;
    Speed_Lift04 : UINT;
    Inputs_Lift03 : ST_MX2\Input;
    Inputs_Lift04 : ST_MX2\Input;
    Status_Lift04 : ST_MX2\Status;
    Commands_Lift04 : ST_MX2\Command;
    N008I0200 : BOOL;
    N008I0201 : BOOL;
    N008I0202 : BOOL;
    N008I0208 : BOOL;
    N008I0209 : BOOL;
    N008I0211 : BOOL;
    N008O0400 : BOOL;
    N008O0405 : BOOL;
    N008O0406 : BOOL;
    N005O406 : BOOL;
    SafetyRelays_Lift03 : BOOL;
    SafetyRelays_Lift04 : BOOL;
    Status_Lift04_Ch : ST_MX2\Status;
    Commands_Lift04_Ch : ST_MX2\Command;
    Speed_Lift04_Ch : UINT;
    N005O401 : BOOL;
    N005O402 : BOOL;
    N005I0209 : BOOL;
    N005I0210 : BOOL;
    N005O403 : BOOL;
    N005I0212 : BOOL;
    N005I0211 : BOOL;
    Freq_Lift04_Ch : UINT;
    N8_Ch1_Counter_Enable : BOOL;
    Led_RS_Extern : BOOL;
    Dummy : BOOL;  (* Dummy *)
    DatAControl_Lift04 : ST_DatAControl_Standard;
    N008I0205 : BOOL;
    N008I0206 : BOOL;
    N008I0213 : BOOL;
    N008I0207 : BOOL;
    N008I0210 : BOOL;
    N008I0301 : BOOL;
    N008I0300 : BOOL;
    N008I0302 : BOOL;
    N008I0303 : BOOL;
    N008I0304 : BOOL;
    N008I0305 : BOOL;
    N008I0306 : BOOL;
    N008I0307 : BOOL;
    N008I0308 : BOOL;
    N008I0309 : BOOL;
    N008I0310 : BOOL;
    N008I0311 : BOOL;
    N008I0312 : BOOL;
    N008I0313 : BOOL;
    N008I0314 : BOOL;
    N008I0315 : BOOL;
    N005I0201 : BOOL;
    N005I0202 : BOOL;
    N005I0309 : BOOL;
    N005I0310 : BOOL;
    N005I0308 : BOOL;
    N005I0311 : BOOL;
    N005O405 : BOOL;
    N005O407 : BOOL;
    N005O400 : BOOL;
    N005O404 : BOOL;
    N008I0203 : BOOL;
    N008I0204 : BOOL;
    N008I0212 : BOOL;
    N008O0407 : BOOL;
    N8_Ch1_Encoder_Preset_Position : DINT;
    N8_Ch1_Preset_Execution : BOOL;
    N8_NX_Unit_I_O_Data_Active_Status : ARRAY[0..63] OF BOOL;
    N8_Ch1_Preset_Command_Value : DINT;
    Comm_From_Carrier01 : ST_FB_40701\Comm_OUT;
    Comm_From_Carrier02 : ST_FB_40701\Comm_OUT;
    Status_Lift03 : ST_MX2\Status;
    Commands_Lift03 : ST_MX2\Command;
    Speed_Lift03 : UINT;
    Freq_Lift03 : UINT;
    Status_Lift03_Ch : ST_MX2\Status;
    Commands_Lift03_Ch : ST_MX2\Command;
    Speed_Lift03_Ch : UINT;
    Freq_Lift03_Ch : UINT;
    Pocket_Lift04 : ST_FB_40401_Commands;
    ES_OK : BOOL;
    TransferBuffer : ST_TransferBuffer;
    Comm_To_Carrier01 : ST_FB_40701\Comm_IN;
    Comm_To_Carrier02 : ST_FB_40701\Comm_IN;
    XTrack_XYPositions_Array : ARRAY[0..199] OF UINT;
    Lift_Array : ARRAY[0..99] OF UINT;
    FixedLoadPosition_Array : ARRAY[0..199] OF UINT;
    FixedUnloadPosition_Array : ARRAY[0..199] OF UINT;
    RegistrationData_Carrier02 : ARRAY[0..199] OF UINT;
    Settings_CP : ST_Settings_CP;
    Area : ARRAY[0..99] OF ST_Area;
    PositionInformation_Rack : ST_FB_40701\PositionInformation_Rack;
    PositionInformation_Rough : ARRAY[0..9] OF UINT;
    XTrack_Y_Values : ARRAY[0..49] OF UDINT;
    PositionInformation_XTrack : ST_FB_40701\PositionInformation_XTrack;
    XTrack : ARRAY[0..49] OF ST_XTrack;
    Grants : ARRAY[0..9999] OF ST_Grant;
    XTrack_X_Values : ARRAY[0..49] OF UDINT;  (* X-Track X values *)
    GrantEnter_Ca01 : BOOL;  (* Grant Enter carrier self *)
    GrantLeave_Ca01 : BOOL;  (* Grant Leave carrier self *)
    ReservationDB : ARRAY[0..20] OF ST_FB_Reservation_Carrier;
    CommSend_Ca01 : BOOL;
    CommReceive_Ca01 : BOOL;
    DstNetAdr_Ca01 : _sDNET_ADR;
    Option_Ca01 : _sRESPONSE;
    Option_Ca02 : _sRESPONSE;
    Comm_To_Carrier02_SENDREC : ARRAY[0..199] OF WORD;
    Comm_From_Carrier02_SENDREC : ARRAY[0..199] OF WORD;
    Comm_To_Carrier01_SENDREC : ARRAY[0..199] OF WORD;
    DstNetAdr_Ca02 : _sDNET_ADR;
    Comm_From_Carrier01_SENDREC : ARRAY[0..199] OF WORD;
    GrantLeave_Ca02 : BOOL;
    CommSend_Ca02 : BOOL;
    CommReceive_Ca02 : BOOL;
    GrantEnter_Ca02 : BOOL;
    N008O0401 : BOOL;  (* Charger_3D105 *)
    N008O0403 : BOOL;
    N008O0404 : BOOL;
    N008O0402 : BOOL;
    N005I0203 : BOOL;
    N005I0205 : BOOL;
    N005I0204 : BOOL;
    N005I0208 : BOOL;
    N005I0206 : BOOL;
    N005I0213 : BOOL;
    N005I0207 : BOOL;
    Lift : ARRAY[0..9] OF ST_LiftInformation;
    Comm_W02_LiftGR04 : ST_FB_25050\CommOutPipe;
    Comm_LiftGR4_W02 : ST_FB_25050\CommInPipe;
    N000O0101 : BOOL;
    N000O0100 : BOOL;
    N005I0300 : BOOL;
    N005I0304 : BOOL;
    N005I0312 : BOOL;
    N005I0313 : BOOL;
    N005I0314 : BOOL;
    N005I0315 : BOOL;
    DatAControl_Lift03 : ST_DatAControl_Standard;
    Pocket_Lift03 : ST_FB_40401_Commands;
    EncoderRackMM : UDINT;
    Speed_Rack_MM_per_Sec : REAL;
    Speed_Rack_M_per_Sec : REAL;
    Speed_Rack_KM_per_Hour : REAL;
    EncoderXtrackMM : UDINT;
    Speed_XTrack_MM_per_Sec : REAL;
    Speed_XTrack_M_per_Sec : REAL;
    Speed_XTrack_KM_per_Hour : REAL;
    N005I0307 : BOOL;
    RegistrationData_Carrier01 : ARRAY[0..199] OF UINT;
    N33_Ch1_Preset_Execution : BOOL;
    N33_Ch1_Encoder_Preset_Position : DINT;
    N33_Ch1_Counter_Enable : BOOL;
    N33_NX_Unit_I_O_Data_Active_Status : ARRAY[0..63] OF BOOL;
    N33_Ch1_Preset_Command_Value : DINT;
    Inputs_Lift03_Ch : ST_MX2\Input;
    Inputs_Lift04_Ch : ST_MX2\Input;
    Comm_LiftGR3_W01 : ST_FB_25050\CommInPipe;
    Comm_W01_LiftGR3 : ST_FB_25050\CommOutPipe;
    LiftGR04NotLoaded : BOOL;
    LiftGR03NotLoaded : BOOL;
    Comm_W07_LiftGR04 : ST_FB_25050\CommOutPipe;
    Comm_LiftGR4_W07 : ST_FB_25050\CommInPipe;
    Comm_W06_LiftGR3 : ST_FB_25050\CommOutPipe;
    Comm_LiftGR3_W06 : ST_FB_25050\CommInPipe;
    Comm_To_Carrier03 : ST_FB_40701\Comm_IN;
    Comm_From_Carrier03 : ST_FB_40701\Comm_OUT;
    RegistrationData_Carrier03 : ARRAY[0..199] OF UINT;
    GrantEnter_Ca03 : BOOL;
    GrantLeave_Ca03 : BOOL;
    DstNetAdr_Ca03 : _sDNET_ADR;
    Option_Ca03 : _sRESPONSE;
    CommReceive_Ca03 : BOOL;
    CommSend_Ca03 : BOOL;
    Comm_To_Carrier03_SENDREC : ARRAY[0..199] OF WORD;
    Comm_From_Carrier03_SENDREC : ARRAY[0..199] OF WORD;
    Comm_LiftGR4_W03 : ST_FB_25050\CommInPipe;
    Comm_LiftGR4_W05 : ST_FB_25050\CommInPipe;
    Comm_W03_LiftGR04 : ST_FB_25050\CommOutPipe;
    Comm_W05_LiftGR04 : ST_FB_25050\CommOutPipe;
    I_EStop_OK : BOOL;
    N005I0214 : BOOL;
    N005I0215 : BOOL;
    N008I0214 : BOOL;
    N008I0215 : BOOL;
    EncoderLift03 : UDINT;  (* Current encoder value of lift 03 *)
    EncoderLift04 : UDINT;  (* Current encoder value of lift 04 *)
    Lift3_PulsValueLevel1 : UDINT;
    Lift3_PulsValueLevel2 : UDINT;
    Lift3_PulsValueLevel3 : UDINT;
    Lift3_PulsValueLevel4 : UDINT;
    Lift3_PulsValueLevel5 : UDINT;
    Lift3_PulsValueLevel6 : UDINT;
    Lift3_PulsValueLevel7 : UDINT;
    Lift3_PulsValueLevel8 : UDINT;
    Lift3_PulsValueLevel9 : UDINT;
    Lift4_PulsValueLevel1 : UDINT;
    Lift4_PulsValueLevel2 : UDINT;
    Lift4_PulsValueLevel3 : UDINT;
    Lift4_PulsValueLevel4 : UDINT;
    Lift4_PulsValueLevel5 : UDINT;
    Lift4_PulsValueLevel6 : UDINT;
    Lift4_PulsValueLevel7 : UDINT;
    Lift4_PulsValueLevel8 : UDINT;
    Lift4_PulsValueLevel9 : UDINT;
    Lift4_PulsValueLevel10 : UDINT;
    Lift3_PulsValueLevel1_Backup : UDINT;
    Lift3_PulsValueLevel2_Backup : UDINT;
    Lift3_PulsValueLevel3_Backup : UDINT;
    Lift3_PulsValueLevel4_Backup : UDINT;
    Lift3_PulsValueLevel5_Backup : UDINT;
    Lift3_PulsValueLevel6_Backup : UDINT;
    Lift3_PulsValueLevel7_Backup : UDINT;
    Lift3_PulsValueLevel8_Backup : UDINT;
    Lift3_PulsValueLevel9_Backup : UDINT;
    Lift4_PulsValueLevel1_Backup : UDINT;
    Lift4_PulsValueLevel2_Backup : UDINT;
    Lift4_PulsValueLevel3_Backup : UDINT;
    Lift4_PulsValueLevel4_Backup : UDINT;
    Lift4_PulsValueLevel5_Backup : UDINT;
    Lift4_PulsValueLevel6_Backup : UDINT;
    Lift4_PulsValueLevel7_Backup : UDINT;
    Lift4_PulsValueLevel9_Backup : UDINT;
    Lift4_PulsValueLevel10_Backup : UDINT;
    Lift4_PulsValueLevel8_Backup : UDINT;
    N000O0103 : BOOL;
    N005I0302 : BOOL;
    N005I0301 : BOOL;
    N005I0303 : BOOL;
    N005I0305 : BOOL;
    Lift3_Extra_Warning1 : WORD;
    Lift3_Extra_Warning2 : WORD;
    Lift4_Extra_Warning1 : WORD;
    Lift4_Extra_Warning2 : WORD;
    LC_Lift3_Disable_Back_Level0 : BOOL;
    LC_Lift3_Disable_Back_Level4 : BOOL;
    LC_Lift3_Disable_Front_Level0 : BOOL;
    LC_Lift3_Disable_Front_Level1 : BOOL;
    LC_Lift3_Disable_Front_Level2 : BOOL;
    LC_Lift3_Disable_Front_Level3 : BOOL;
    LC_Lift3_Disable_Front_Level4 : BOOL;
    LC_Lift3_Disable_Front_Level5 : BOOL;
    LC_Lift3_Disable_Front_Level6 : BOOL;
    LC_Lift3_Disable_Front_Level7 : BOOL;
    LC_LIft4_Disable_Back_Level0 : BOOL;
    LC_LIft4_Disable_Back_Level4 : BOOL;
    LC_LIft4_Disable_Front_Level0 : BOOL;
    LC_LIft4_Disable_Front_Level1 : BOOL;
    LC_LIft4_Disable_Front_Level2 : BOOL;
    LC_LIft4_Disable_Front_Level3 : BOOL;
    LC_LIft4_Disable_Front_Level4 : BOOL;
    LC_LIft4_Disable_Front_Level5 : BOOL;
    LC_LIft4_Disable_Front_Level6 : BOOL;
    LC_LIft4_Disable_Front_Level7 : BOOL;
    Lift4_Extra_Warning3 : WORD;
    Lift3_Extra_Warning3 : WORD;
    WarningBadCommC1 : BOOL;
    WarningBadCommC2 : BOOL;
    WarningBadCommC3 : BOOL;
    Comm_To_Carrier04 : ST_FB_40701\Comm_IN;
    Comm_From_Carrier04 : ST_FB_40701\Comm_OUT;
    WarningBadCommC4 : BOOL;
    RegistrationData_Carrier04 : ARRAY[0..199] OF UINT;
    GrantEnter_Ca04 : BOOL;
    GrantLeave_Ca04 : BOOL;
    CommSend_Ca04 : BOOL;
    CommReceive_Ca04 : BOOL;
    DstNetAdr_Ca04 : _sDNET_ADR;
    Option_Ca04 : _sRESPONSE;
    Comm_To_Carrier04_SENDREC : ARRAY[0..199] OF WORD;
    Comm_From_Carrier04_SENDREC : ARRAY[0..199] OF WORD;
    Comm_To_Carrier05 : ST_FB_40701\Comm_IN;
    Comm_From_Carrier05 : ST_FB_40701\Comm_OUT;
    WarningBadCommC5 : BOOL;
    RegistrationData_Carrier05 : ARRAY[0..199] OF UINT;
    GrantEnter_Ca05 : BOOL;
    GrantLeave_Ca05 : BOOL;
    CommSend_Ca05 : BOOL;
    CommReceive_Ca05 : BOOL;
    DstNetAdr_Ca05 : _sDNET_ADR;
    Comm_To_Carrier05_SENDREC : ARRAY[0..199] OF WORD;
    Option_Ca05 : _sRESPONSE;
    Comm_From_Carrier05_SENDREC : ARRAY[0..199] OF WORD;
    N000O0104 : BOOL;  (* Charger_4D105 *)
    N000O0105 : BOOL;
    N05_Major_Fault : BOOL;
    N05_Minor_Fault : BOOL;
    N05_Partial_Fault : BOOL;
    N33_Major_Fault : BOOL;
    N33_Minor_Fault : BOOL;
    N33_Partial_Fault : BOOL;
    N08_Major_Fault : BOOL;
    N08_Minor_Fault : BOOL;
    N08_Partial_Fault : BOOL;
    N43_Major_Fault : BOOL;
    N43_Minor_Fault : BOOL;
    N43_Partial_Fault : BOOL;
    Lift03_Status : ST_FB_40401_Status;
    Lift04_Status : ST_FB_40401_Status;
    Charger4D105_DatAControl : ST_DatAControl_Standard;
    Commands_Charger4D105 : ST_FB_1xxxx\FB_10001_Commands;
    Commands_Charger3D105 : ST_FB_1xxxx\FB_10001_Commands;
    Charger3D105_DatAControl : ST_DatAControl_Standard;
    Charger4D402_DatAControl : ST_DatAControl_Standard;
    Commands_Charger4D402 : ST_FB_1xxxx\FB_10001_Commands;
    Charger4D102_DatAControl : ST_DatAControl_Standard;
    Commands_Charger4D102 : ST_FB_1xxxx\FB_10001_Commands;
    Charger3D202_DatAControl : ST_DatAControl_Standard;
    Commands_Charger3D202 : ST_FB_1xxxx\FB_10001_Commands;
END_VAR
VAR
    _p1 : BOOL;
    _t2 : BOOL;
    _p3 : BOOL;
    _t4 : BOOL;
    _e5 : R_TRIG;
    _p6 : BOOL;
    _e7 : R_TRIG;
    _p8 : BOOL;
    _t9 : BOOL;
    _p10 : BOOL;
    _e11 : R_TRIG;
    _e12 : R_TRIG;
    _e13 : R_TRIG;
    _e14 : R_TRIG;
    _p15 : BOOL;
    _t16 : BOOL;
    _p17 : BOOL;
    _t18 : BOOL;
    _e19 : R_TRIG;
    _p20 : BOOL;
    _e21 : R_TRIG;
    _p22 : BOOL;
    _t23 : BOOL;
    _p24 : BOOL;
    _e25 : R_TRIG;
    _e26 : R_TRIG;
    _e27 : R_TRIG;
    _e28 : R_TRIG;
    _p29 : BOOL;
    _t30 : BOOL;
    _p31 : BOOL;
    _t32 : BOOL;
    _e33 : R_TRIG;
    _p34 : BOOL;
    _e35 : R_TRIG;
    _p36 : BOOL;
    _t37 : BOOL;
    _p38 : BOOL;
    _e39 : R_TRIG;
    _e40 : R_TRIG;
    _e41 : R_TRIG;
    _e42 : R_TRIG;
    _p43 : BOOL;
    _t44 : BOOL;
    _p45 : BOOL;
    _t46 : BOOL;
    _e47 : R_TRIG;
    _p48 : BOOL;
    _e49 : R_TRIG;
    _p50 : BOOL;
    _t51 : BOOL;
    _p52 : BOOL;
    _e53 : R_TRIG;
    _e54 : R_TRIG;
    _e55 : R_TRIG;
    _e56 : R_TRIG;
    _p57 : BOOL;
    _t58 : BOOL;
    _p59 : BOOL;
    _t60 : BOOL;
    _e61 : R_TRIG;
    _p62 : BOOL;
    _e63 : R_TRIG;
    _p64 : BOOL;
    _t65 : BOOL;
    _p66 : BOOL;
    _e67 : R_TRIG;
    _e68 : R_TRIG;
    _e69 : R_TRIG;
    _e70 : R_TRIG;
END_VAR

(* Section Lift03: ladder, written here as Structured Text *)

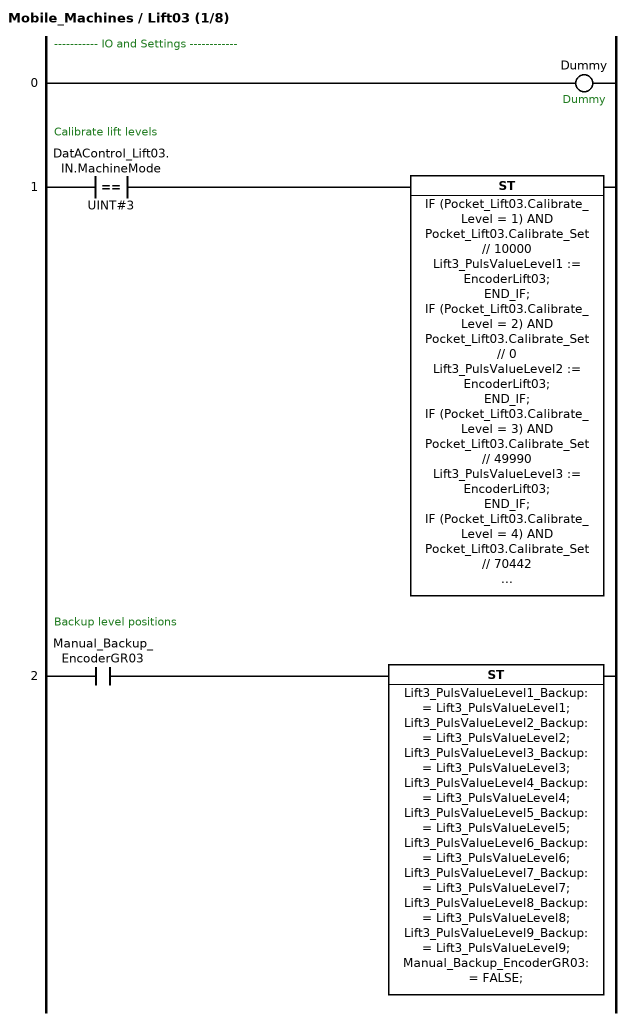
(* Rung 0: ----------- IO and Settings ------------ *)
Dummy := TRUE;
(* Rung 1: Calibrate lift levels *)
IF DatAControl_Lift03.IN.MachineMode = UINT#3 THEN
    IF (Pocket_Lift03.Calibrate_Level = 1) AND Pocket_Lift03.Calibrate_SetLevel THEN
    	// 10000
    	Lift3_PulsValueLevel1 := EncoderLift03;
    END_IF;
    
    IF (Pocket_Lift03.Calibrate_Level = 2) AND Pocket_Lift03.Calibrate_SetLevel THEN
    	// 0
    	Lift3_PulsValueLevel2 := EncoderLift03;
    END_IF;
    
    IF (Pocket_Lift03.Calibrate_Level = 3) AND Pocket_Lift03.Calibrate_SetLevel THEN
    	// 49990
    	Lift3_PulsValueLevel3 := EncoderLift03;
    END_IF;
    
    IF (Pocket_Lift03.Calibrate_Level = 4) AND Pocket_Lift03.Calibrate_SetLevel THEN
    	// 70442
    	Lift3_PulsValueLevel4 := EncoderLift03;
    END_IF;
    
    IF (Pocket_Lift03.Calibrate_Level = 5) AND Pocket_Lift03.Calibrate_SetLevel THEN
    	//90882
    	Lift3_PulsValueLevel5 := EncoderLift03;
    END_IF;
    
    IF (Pocket_Lift03.Calibrate_Level = 6) AND Pocket_Lift03.Calibrate_SetLevel THEN
    	// 111334
    	Lift3_PulsValueLevel6 := EncoderLift03;
    END_IF;
    
    IF (Pocket_Lift03.Calibrate_Level = 7) AND Pocket_Lift03.Calibrate_SetLevel THEN
    	// 131808
    	Lift3_PulsValueLevel7 := EncoderLift03;
    END_IF;
    
    IF (Pocket_Lift03.Calibrate_Level = 8) AND Pocket_Lift03.Calibrate_SetLevel THEN
    	// 152225
    	Lift3_PulsValueLevel8 := EncoderLift03;
    END_IF;
    
    IF (Pocket_Lift03.Calibrate_Level = 9) AND Pocket_Lift03.Calibrate_SetLevel THEN
    	// 172672
    	Lift3_PulsValueLevel9 := EncoderLift03;
    END_IF;
    
    Pocket_Lift03.Calibrate_SetLevel := FALSE;
END_IF;
(* Rung 2: Backup level positions *)
IF Manual_Backup_EncoderGR03 THEN
    Lift3_PulsValueLevel1_Backup:= Lift3_PulsValueLevel1;
    Lift3_PulsValueLevel2_Backup:= Lift3_PulsValueLevel2;
    Lift3_PulsValueLevel3_Backup:= Lift3_PulsValueLevel3;
    Lift3_PulsValueLevel4_Backup:= Lift3_PulsValueLevel4;
    Lift3_PulsValueLevel5_Backup:= Lift3_PulsValueLevel5;
    Lift3_PulsValueLevel6_Backup:= Lift3_PulsValueLevel6;
    Lift3_PulsValueLevel7_Backup:= Lift3_PulsValueLevel7;
    Lift3_PulsValueLevel8_Backup:= Lift3_PulsValueLevel8;
    Lift3_PulsValueLevel9_Backup:= Lift3_PulsValueLevel9;
    
    Manual_Backup_EncoderGR03:= FALSE;
END_IF;

